      ;FOLD -- RSK Sammelstoerung -- ;%{SE}%MKUKATPVW %CVW_COM %VCOMMENT %P 2:-- RSK Sammelstoerung --, 3: VW_COMMENT
      ;ENDFOLD
      ;FOLD F329 = T7 + T9 + F325 ;%{SE}%MKUKATPVW %CVW_SPS %VBOASG %P 2:F329 = T7 + T9 + F325, 3: BOASG
         $FLAG[329] = $TIMER_FLAG[7] OR $TIMER_FLAG[9] OR $FLAG[325]
      ;ENDFOLD
      ;FOLD -- Hilfsflag Startfraesen -- ;%{SE}%MKUKATPVW %CVW_COM %VCOMMENT %P 2:-- Hilfsflag Startfraesen --, 3: VW_COMMENT
      ;ENDFOLD
      ;FOLD F152 = (F152 & F138 + F154 & F139) & F287 ;%{SE}%MKUKATPVW %CVW_SPS %VBOASG %P 2:F152 = (F152 & F138 + F154 & F139) & F287, 3: BOASG
         $FLAG[152] = ($FLAG[152] AND $FLAG[138] OR $FLAG[154] AND $FLAG[139]) AND $FLAG[287]
      ;ENDFOLD
      ;FOLD F154 = !F164 & F154 + F164 & F287 & F154 ;%{SE}%MKUKATPVW %CVW_SPS %VBOASG %P 2:F154 = !F164 & F154 + F164 & F287 & F154, 3: BOASG
         $FLAG[154] = NOT $FLAG[164] AND $FLAG[154] OR $FLAG[164] AND $FLAG[287] AND $FLAG[154]
      ;ENDFOLD
      ;FOLD F287 = F138 + F139 & F164 ;%{SE}%MKUKATPVW %CVW_SPS %VBOASG %P 2:F287 = F138 + F139 & F164, 3: BOASG
         $FLAG[287] = $FLAG[138] OR $FLAG[139] AND $FLAG[164]
      ;ENDFOLD
      ;FOLD -- Neues Fraesprogramm und Zaehler ruecksetzen -- ;%{SE}%MKUKATPVW %CVW_COM %VCOMMENT %P 2:-- Neues Fraesprogramm und Zaehler ruecksetzen --, 3: VW_COMMENT
      ;ENDFOLD
      ;FOLD bin3 ( F164 ) = 36 ;%{SE}%MKUKATPVW %CVW_SPS %VARIASG %P 2:bin3 ( F164 ) = 36, 3: ARIASG
         VW(#BINOUT,$FLAG[164],3,36)
      ;ENDFOLD
      ;FOLD i7 ( F152 ) = i45 ;%{SE}%MKUKATPVW %CVW_SPS %VARIASG %P 2:i7 ( F152 ) = i45, 3: ARIASG
         VW(#COUNTER,$FLAG[152],7,$COUNT_I[45])
      ;ENDFOLD
      ;FOLD -- Wiederholung beim Startfraesen -- ;%{SE}%MKUKATPVW %CVW_COM %VCOMMENT %P 2:-- Wiederholung beim Startfraesen --, 3: VW_COMMENT
      ;ENDFOLD
      ;FOLD Schritt 81 = E877 & !E878 & (F138 & !F152 + F139 & F164 & !F152) & !F325 & !F329 & A4039 ;%{SE}%MKUKATPVW %CVW_SPS %VST_CON %P 2:Schritt 81 = E877 & !E878 & (F138 & !F152 + F139 & F164 & !F152) & !F325 & !F329 & A4039, 3: ST_CON
         IF $IN[877] AND NOT $IN[878] AND ($FLAG[138] AND NOT $FLAG[152] OR $FLAG[139] AND $FLAG[164] AND NOT $FLAG[152]) AND NOT $FLAG[325] AND NOT $FLAG[329] AND $OUT[4039] THEN
            PREVSTEP = $APP_INT[5]
            $APP_INT[5] = 81
         ENDIF
      ;ENDFOLD
      ;FOLD -- Weiter wenn Fraesen fertig -- ;%{SE}%MKUKATPVW %CVW_COM %VCOMMENT %P 2:-- Weiter wenn Fraesen fertig --, 3: VW_COMMENT
      ;ENDFOLD
      ;FOLD Schritt 85 = E877 & !E878 & (F139 & F154 & (!F164 + F152) + F138 & F152 + F325 + F329) & A4039 ;%{SE}%MKUKATPVW %CVW_SPS %VST_CON %P 2:Schritt 85 = E877 & !E878 & (F139 & F154 & (!F164 + F152) + F138 & F152 + F325 + F329) & A4039, 3: ST_CON
         IF $IN[877] AND NOT $IN[878] AND ($FLAG[139] AND $FLAG[154] AND (NOT $FLAG[164] OR $FLAG[152]) OR $FLAG[138] AND $FLAG[152] OR $FLAG[325] OR $FLAG[329]) AND $OUT[4039] THEN
            PREVSTEP = $APP_INT[5]
            $APP_INT[5] = 85
         ENDIF
      ;ENDFOLD
   ;ENDFOLD
   ;FOLD SCHRITT 85 -- STAT EZ2/SP2/KE2-- ;%{P}%MKUKATPVW,%CSTEP,%VST_NR,%P 1:SCHRITT, 2:85, 3: STAT EZ2/SP2/KE2
      ;FOLD ;%{H}
         Case 85
      ;ENDFOLD
      ;FOLD F324 = AUS ;%{SE}%MKUKATPVW %CVW_SPS %VBOASG %P 2:F324 = AUS, 3: BOASG
         $FLAG[324] = FALSE
      ;ENDFOLD
      ;FOLD A877 = AUS ;%{SE}%MKUKATPVW %CVW_SPS %VBOASG %P 2:A877 = AUS, 3: BOASG
         $OUT[877] = FALSE
      ;ENDFOLD
      ;FOLD -- KF2 abschalten -- ;%{SE}%MKUKATPVW %CVW_COM %VCOMMENT %P 2:-- KF2 abschalten --, 3: VW_COMMENT
      ;ENDFOLD
      ;FOLD A994 = AUS ;%{SE}%MKUKATPVW %CVW_SPS %VBOASG %P 2:A994 = AUS, 3: BOASG
         $OUT[994] = FALSE
      ;ENDFOLD
      ;FOLD -- Ueberwachungszeit KF2 Versetzeinheit -- ;%{SE}%MKUKATPVW %CVW_COM %VCOMMENT %P 2:-- Ueberwachungszeit KF2 Versetzeinheit --, 3: VW_COMMENT
      ;ENDFOLD
      ;FOLD t8 ( EIN ) = -40[1/10Sek] ;%{SE}%MKUKATPVW %CVW_SPS %VTASG %P 2:t8 ( EIN ) = -40[1/10Sek], 3: TASG
         VW(#SET_TIME,TRUE,8,0,-40)
      ;ENDFOLD
      ;FOLD Schritt 86 = A4039 ;%{SE}%MKUKATPVW %CVW_SPS %VST_CON %P 2:Schritt 86 = A4039, 3: ST_CON
         IF $OUT[4039] THEN
            PREVSTEP = $APP_INT[5]
            $APP_INT[5] = 86
         ENDIF
      ;ENDFOLD
   ;ENDFOLD
   ;FOLD SCHRITT 86 -- STAT EZ2/SP2/KE2 -- ;%{P}%MKUKATPVW,%CSTEP,%VST_NR,%P 1:SCHRITT, 2:86, 3: STAT EZ2/SP2/KE2
      ;FOLD ;%{H}
         Case 86
      ;ENDFOLD
      ;FOLD F328 = AUS ;%{SE}%MKUKATPVW %CVW_SPS %VBOASG %P 2:F328 = AUS, 3: BOASG
         $FLAG[328] = FALSE
      ;ENDFOLD
      ;FOLD -- KF2 Versetzeinheit vor -- ;%{SE}%MKUKATPVW %CVW_COM %VCOMMENT %P 2:-- KF2 Versetzeinheit vor --, 3: VW_COMMENT
      ;ENDFOLD
      ;FOLD A995 = F565 ;%{SE}%MKUKATPVW %CVW_SPS %VBOASG %P 2:A995 = F565, 3: BOASG
         $OUT[995] = $FLAG[565]
      ;ENDFOLD
      ;FOLD -- RSK Fehlerausgabe KS2 Arbeitsst. -- ;%{SE}%MKUKATPVW %CVW_COM %VCOMMENT %P 2:-- RSK Fehlerausgabe KS2 Arbeitsst. --, 3: VW_COMMENT
      ;ENDFOLD
      ;FOLD F324 = (E996 + !E997 + !E998 + E999) & !F323 & !F328 + F324 ;%{SE}%MKUKATPVW %CVW_SPS %VBOASG %P 2:F324 = (E996 + !E997 + !E998 + E999) & !F323 & !F328 + F324, 3: BOASG
         $FLAG[324] = ($IN[996] OR NOT $IN[997] OR NOT $IN[998] OR $IN[999]) AND NOT $FLAG[323] AND NOT $FLAG[328] OR $FLAG[324]
      ;ENDFOLD
      ;FOLD -- RSK Sammelstoerung -- ;%{SE}%MKUKATPVW %CVW_COM %VCOMMENT %P 2:-- RSK Sammelstoerung --, 3: VW_COMMENT
      ;ENDFOLD
      ;FOLD F329 = F324 + F325 ;%{SE}%MKUKATPVW %CVW_SPS %VBOASG %P 2:F329 = F324 + F325, 3: BOASG
         $FLAG[329] = $FLAG[324] OR $FLAG[325]
      ;ENDFOLD
      ;FOLD -- Ueberwachungszeit KS2 schwenken -- ;%{SE}%MKUKATPVW %CVW_COM %VCOMMENT %P 2:-- Ueberwachungszeit KS2 schwenken --, 3: VW_COMMENT
      ;ENDFOLD
      ;FOLD t9 ( EIN ) = -100[1/10Sek] ;%{SE}%MKUKATPVW %CVW_SPS %VTASG %P 2:t9 ( EIN ) = -100[1/10Sek], 3: TASG
         VW(#SET_TIME,TRUE,9,0,-100)
      ;ENDFOLD
      ;FOLD Schritt 85 = F324 & (E26 + E27) & A4039 ;%{SE}%MKUKATPVW %CVW_SPS %VST_CON %P 2:Schritt 85 = F324 & (E26 + E27) & A4039, 3: ST_CON
         IF $FLAG[324] AND ($IN[26] OR $IN[27]) AND $OUT[4039] THEN
            PREVSTEP = $APP_INT[5]
            $APP_INT[5] = 85
         ENDIF
      ;ENDFOLD
      ;FOLD Schritt 87 = (!F324 & (E995 & F565 + !E995 & !F565) + T8 + F325) & A4039 ;%{SE}%MKUKATPVW %CVW_SPS %VST_CON %P 2:Schritt 87 = (!F324 & (E995 & F565 + !E995 & !F565) + T8 + F325) & A4039, 3: ST_CON
         IF (NOT $FLAG[324] AND ($IN[995] AND $FLAG[565] OR NOT $IN[995] AND NOT $FLAG[565]) OR $TIMER_FLAG[8] OR $FLAG[325]) AND $OUT[4039] THEN
            PREVSTEP = $APP_INT[5]
            $APP_INT[5] = 87
         ENDIF
      ;ENDFOLD
   ;ENDFOLD
   ;FOLD SCHRITT 87 -- STAT EZ2/SP2/KE2-- ;%{P}%MKUKATPVW,%CSTEP,%VST_NR,%P 1:SCHRITT, 2:87, 3: STAT EZ2/SP2/KE2
      ;FOLD ;%{H}
         Case 87
      ;ENDFOLD
      ;FOLD F323 = AUS ;%{SE}%MKUKATPVW %CVW_SPS %VBOASG %P 2:F323 = AUS, 3: BOASG
         $FLAG[323] = FALSE
      ;ENDFOLD
      ;FOLD F328 = AUS ;%{SE}%MKUKATPVW %CVW_SPS %VBOASG %P 2:F328 = AUS, 3: BOASG
         $FLAG[328] = FALSE
      ;ENDFOLD
      ;FOLD -- RSK Sammelstoerung -- ;%{SE}%MKUKATPVW %CVW_COM %VCOMMENT %P 2:-- RSK Sammelstoerung --, 3: VW_COMMENT
      ;ENDFOLD
      ;FOLD F329 = F325 ;%{SE}%MKUKATPVW %CVW_SPS %VBOASG %P 2:F329 = F325, 3: BOASG
         $FLAG[329] = $FLAG[325]
      ;ENDFOLD
      ;FOLD -- KF2 ein -- ;%{SE}%MKUKATPVW %CVW_COM %VCOMMENT %P 2:-- KF2 ein --, 3: VW_COMMENT
      ;ENDFOLD
      ;FOLD A994 = EIN ;%{SE}%MKUKATPVW %CVW_SPS %VBOASG %P 2:A994 = EIN, 3: BOASG
         $OUT[994] = TRUE
      ;ENDFOLD
      ;FOLD -- KS2 in Ruhestellung schwenken -- ;%{SE}%MKUKATPVW %CVW_COM %VCOMMENT %P 2:-- KS2 in Ruhestellung schwenken --, 3: VW_COMMENT
      ;ENDFOLD
      ;FOLD A1000 = (F746 + !F714) & E877 & (E995 & F565 + !E995 & !F565) ;%{SE}%MKUKATPVW %CVW_SPS %VBOASG %P 2:A1000 = (F746 + !F714) & E877 & (E995 & F565 + !E995 & !F565), 3: BOASG
         $OUT[1000] = ($FLAG[746] OR NOT $FLAG[714]) AND $IN[877] AND ($IN[995] AND $FLAG[565] OR NOT $IN[995] AND NOT $FLAG[565])
      ;ENDFOLD
      ;FOLD Schritt 88 = (F746 + !F714 + T9) & (A1000 + T9) & E877 & A4039 ;%{SE}%MKUKATPVW %CVW_SPS %VST_CON %P 2:Schritt 88 = (F746 + !F714 + T9) & (A1000 + T9) & E877 & A4039, 3: ST_CON
         IF ($FLAG[746] OR NOT $FLAG[714] OR $TIMER_FLAG[9]) AND ($OUT[1000] OR $TIMER_FLAG[9]) AND $IN[877] AND $OUT[4039] THEN
            PREVSTEP = $APP_INT[5]
            $APP_INT[5] = 88
         ENDIF
      ;ENDFOLD
   ;ENDFOLD
   ;FOLD SCHRITT 88 -- STAT EZ2/SP2/KE2 -- ;%{P}%MKUKATPVW,%CSTEP,%VST_NR,%P 1:SCHRITT, 2:88, 3: STAT EZ2/SP2/KE2
      ;FOLD ;%{H}
         Case 88
      ;ENDFOLD
      ;FOLD -- Hilfsflag SK Programmwechsel -- ;%{SE}%MKUKATPVW %CVW_COM %VCOMMENT %P 2:-- Hilfsflag SK Programmwechsel --, 3: VW_COMMENT
      ;ENDFOLD
      ;FOLD F334 = AUS ;%{SE}%MKUKATPVW %CVW_SPS %VBOASG %P 2:F334 = AUS, 3: BOASG
         $FLAG[334] = FALSE
      ;ENDFOLD
      ;FOLD -- RSK Fehlerausgabe KF Versetzeinheit -- ;%{SE}%MKUKATPVW %CVW_COM %VCOMMENT %P 2:-- RSK Fehlerausgabe KF Versetzeinheit --, 3: VW_COMMENT
      ;ENDFOLD
      ;FOLD F328 = !E995 & F565 & !F323 + F328 ;%{SE}%MKUKATPVW %CVW_SPS %VBOASG %P 2:F328 = !E995 & F565 & !F323 + F328, 3: BOASG
         $FLAG[328] = NOT $IN[995] AND $FLAG[565] AND NOT $FLAG[323] OR $FLAG[328]
      ;ENDFOLD
      ;FOLD -- RSK Fehlerausgabe KS2 Ruhestellung -- ;%{SE}%MKUKATPVW %CVW_COM %VCOMMENT %P 2:-- RSK Fehlerausgabe KS2 Ruhestellung --, 3: VW_COMMENT
      ;ENDFOLD
      ;FOLD F323 = (!E996 + E997 + E998 + !E999) & T9 & (E995 + !F565) + F323 ;%{SE}%MKUKATPVW %CVW_SPS %VBOASG %P 2:F323 = (!E996 + E997 + E998 + !E999) & T9 & (E995 + !F565) + F323, 3: BOASG
         $FLAG[323] = (NOT $IN[996] OR $IN[997] OR $IN[998] OR NOT $IN[999]) AND $TIMER_FLAG[9] AND ($IN[995] OR NOT $FLAG[565]) OR $FLAG[323]
      ;ENDFOLD
      ;FOLD -- RSK Fehlerausgabe EZ/SP min. Oeffnung -- ;%{SE}%MKUKATPVW %CVW_COM %VCOMMENT %P 2:-- RSK Fehlerausgabe EZ/SP min. Oeffnung --, 3: VW_COMMENT
      ;ENDFOLD
      ;FOLD F333 = !F746 ;%{SE}%MKUKATPVW %CVW_SPS %VBOASG %P 2:F333 = !F746, 3: BOASG
         $FLAG[333] = NOT $FLAG[746]
      ;ENDFOLD
      ;FOLD -- RSK Sammelstoerung -- ;%{SE}%MKUKATPVW %CVW_COM %VCOMMENT %P 2:-- RSK Sammelstoerung --, 3: VW_COMMENT
      ;ENDFOLD
      ;FOLD F329 = F323 + F325 + F328 + F333 ;%{SE}%MKUKATPVW %CVW_SPS %VBOASG %P 2:F329 = F323 + F325 + F328 + F333, 3: BOASG
         $FLAG[329] = $FLAG[323] OR $FLAG[325] OR $FLAG[328] OR $FLAG[333]
      ;ENDFOLD
      ;FOLD A994 = !F323 & !F328 ;%{SE}%MKUKATPVW %CVW_SPS %VBOASG %P 2:A994 = !F323 & !F328, 3: BOASG
         $OUT[994] = NOT $FLAG[323] AND NOT $FLAG[328]
      ;ENDFOLD
      ;FOLD A995 = F565 ;%{SE}%MKUKATPVW %CVW_SPS %VBOASG %P 2:A995 = F565, 3: BOASG
         $OUT[995] = $FLAG[565]
      ;ENDFOLD
      ;FOLD Schritt 86 = (F323 + F328) & (E26 + E27) & A4039 ;%{SE}%MKUKATPVW %CVW_SPS %VST_CON %P 2:Schritt 86 = (F323 + F328) & (E26 + E27) & A4039, 3: ST_CON
         IF ($FLAG[323] OR $FLAG[328]) AND ($IN[26] OR $IN[27]) AND $OUT[4039] THEN
            PREVSTEP = $APP_INT[5]
            $APP_INT[5] = 86
         ENDIF
      ;ENDFOLD
      ;FOLD Schritt 89 = !A1000 & E996 & !E997 & !E998 & E999 & A4039 ;%{SE}%MKUKATPVW %CVW_SPS %VST_CON %P 2:Schritt 89 = !A1000 & E996 & !E997 & !E998 & E999 & A4039, 3: ST_CON
         IF NOT $OUT[1000] AND $IN[996] AND NOT $IN[997] AND NOT $IN[998] AND $IN[999] AND $OUT[4039] THEN
            PREVSTEP = $APP_INT[5]
            $APP_INT[5] = 89
         ENDIF
      ;ENDFOLD
   ;ENDFOLD
   ;FOLD SCHRITT 89 -- STAT EZ2/SP2/KE2 -- ;%{P}%MKUKATPVW,%CSTEP,%VST_NR,%P 1:SCHRITT, 2:89, 3: STAT EZ2/SP2/KE2
      ;FOLD ;%{H}
         Case 89
      ;ENDFOLD
      ;FOLD F323 = AUS ;%{SE}%MKUKATPVW %CVW_SPS %VBOASG %P 2:F323 = AUS, 3: BOASG
         $FLAG[323] = FALSE
      ;ENDFOLD
      ;FOLD F328 = AUS ;%{SE}%MKUKATPVW %CVW_SPS %VBOASG %P 2:F328 = AUS, 3: BOASG
         $FLAG[328] = FALSE
      ;ENDFOLD
      ;FOLD -- RSK Sammelstoerung -- ;%{SE}%MKUKATPVW %CVW_COM %VCOMMENT %P 2:-- RSK Sammelstoerung --, 3: VW_COMMENT
      ;ENDFOLD
      ;FOLD F329 = F325 ;%{SE}%MKUKATPVW %CVW_SPS %VBOASG %P 2:F329 = F325, 3: BOASG
         $FLAG[329] = $FLAG[325]
      ;ENDFOLD
      ;FOLD t9 ( EIN ) = STOP ;%{SE}%MKUKATPVW %CVW_SPS %VTSTOP %P 2:t9 ( EIN ) = STOP, 3: TSTOP
         VW(#SET_TIME,TRUE,9,1,0)
      ;ENDFOLD
      ;FOLD -- KF2 Versetzeinheit rueck -- ;%{SE}%MKUKATPVW %CVW_COM %VCOMMENT %P 2:-- KF2 Versetzeinheit rueck --, 3: VW_COMMENT
      ;ENDFOLD
      ;FOLD A995 = AUS ;%{SE}%MKUKATPVW %CVW_SPS %VBOASG %P 2:A995 = AUS, 3: BOASG
         $OUT[995] = FALSE
      ;ENDFOLD
      ;FOLD -- KF2 aus -- ;%{SE}%MKUKATPVW %CVW_COM %VCOMMENT %P 2:-- KF2 aus --, 3: VW_COMMENT
      ;ENDFOLD
      ;FOLD A994 = AUS ;%{SE}%MKUKATPVW %CVW_SPS %VBOASG %P 2:A994 = AUS, 3: BOASG
         $OUT[994] = FALSE
      ;ENDFOLD
      ;FOLD -- KF1 Ausblasen -- ;%{SE}%MKUKATPVW %CVW_COM %VCOMMENT %P 2:-- KF1 Ausblasen --, 3: VW_COMMENT
      ;ENDFOLD
      ;FOLD A996 = (F330 + F331 + F332) & F738 ;%{SE}%MKUKATPVW %CVW_SPS %VBOASG %P 2:A996 = (F330 + F331 + F332) & F738, 3: BOASG
         $OUT[996] = ($FLAG[330] OR $FLAG[331] OR $FLAG[332]) AND $FLAG[738]
      ;ENDFOLD
      ;FOLD bin3 ( F285 ) = 5 ;%{SE}%MKUKATPVW %CVW_SPS %VARIASG %P 2:bin3 ( F285 ) = 5, 3: ARIASG
         VW(#BINOUT,$FLAG[285],3,5)
      ;ENDFOLD
      ;FOLD bin6 ( !F285 ) = 1 ;%{SE}%MKUKATPVW %CVW_SPS %VARIASG %P 2:bin6 ( !F285 ) = 1, 3: ARIASG
         VW(#BINOUT,NOT $FLAG[285],6,1)
      ;ENDFOLD
      ;FOLD -- Wartezeit Programmwechsel SK -- ;%{SE}%MKUKATPVW %CVW_COM %VCOMMENT %P 2:-- Wartezeit Programmwechsel SK --, 3: VW_COMMENT
      ;ENDFOLD
      ;FOLD T8 ( !F334 ) = -2[1/10Sek] ;%{SE}%MKUKATPVW %CVW_SPS %VTASG %P 2:T8 ( !F334 ) = -2[1/10Sek], 3: TASG
         VW(#SET_TIME,NOT $FLAG[334],8,0,-2)
      ;ENDFOLD
      ;FOLD -- Hilfsflag SK Programmwechsel -- ;%{SE}%MKUKATPVW %CVW_COM %VCOMMENT %P 2:-- Hilfsflag SK Programmwechsel --, 3: VW_COMMENT
      ;ENDFOLD
      ;FOLD F334 = EIN ;%{SE}%MKUKATPVW %CVW_SPS %VBOASG %P 2:F334 = EIN, 3: BOASG
         $FLAG[334] = TRUE
      ;ENDFOLD
      ;FOLD -- Ueberwachungszeit EZ2/SP2/KE2 Messen -- ;%{SE}%MKUKATPVW %CVW_COM %VCOMMENT %P 2:-- Ueberwachungszeit EZ2/SP2/KE2 Messen --, 3: VW_COMMENT
      ;ENDFOLD
      ;FOLD t9 ( EIN ) = -150[1/10Sek] ;%{SE}%MKUKATPVW %CVW_SPS %VTASG %P 2:t9 ( EIN ) = -150[1/10Sek], 3: TASG
         VW(#SET_TIME,TRUE,9,0,-150)
      ;ENDFOLD
      ;FOLD Schritt 74 = (F325 + F329) & (E26 + E27) & A4039 ;%{SE}%MKUKATPVW %CVW_SPS %VST_CON %P 2:Schritt 74 = (F325 + F329) & (E26 + E27) & A4039, 3: ST_CON
         IF ($FLAG[325] OR $FLAG[329]) AND ($IN[26] OR $IN[27]) AND $OUT[4039] THEN
            PREVSTEP = $APP_INT[5]
            $APP_INT[5] = 74
         ENDIF
      ;ENDFOLD
      ;FOLD Schritt 90 = T8 & !F325 & !F329 & A4039 ;%{SE}%MKUKATPVW %CVW_SPS %VST_CON %P 2:Schritt 90 = T8 & !F325 & !F329 & A4039, 3: ST_CON
         IF $TIMER_FLAG[8] AND NOT $FLAG[325] AND NOT $FLAG[329] AND $OUT[4039] THEN
            PREVSTEP = $APP_INT[5]
            $APP_INT[5] = 90
         ENDIF
      ;ENDFOLD
   ;ENDFOLD
   ;FOLD SCHRITT 90 -- STAT EZ2/SP2/KE2 -- ;%{P}%MKUKATPVW,%CSTEP,%VST_NR,%P 1:SCHRITT, 2:90, 3: STAT EZ2/SP2/KE2
      ;FOLD ;%{H}
         Case 90
      ;ENDFOLD
      ;FOLD -- Hilfsflag SK Programmwechsel -- ;%{SE}%MKUKATPVW %CVW_COM %VCOMMENT %P 2:-- Hilfsflag SK Programmwechsel --, 3: VW_COMMENT
      ;ENDFOLD
      ;FOLD F334 = AUS ;%{SE}%MKUKATPVW %CVW_SPS %VBOASG %P 2:F334 = AUS, 3: BOASG
         $FLAG[334] = FALSE
      ;ENDFOLD
      ;FOLD -- Quitt. Fraesen SK2/SK1 -- ;%{SE}%MKUKATPVW %CVW_COM %VCOMMENT %P 2:-- Quitt. Fraesen SK2/SK1 --, 3: VW_COMMENT
      ;ENDFOLD
      ;FOLD A946 = !F285 & !F329 & !F322 ;%{SE}%MKUKATPVW %CVW_SPS %VBOASG %P 2:A946 = !F285 & !F329 & !F322, 3: BOASG
         $OUT[946] = NOT $FLAG[285] AND NOT $FLAG[329] AND NOT $FLAG[322]
      ;ENDFOLD
      ;FOLD A786 = F285 & !F329 & !F322 ;%{SE}%MKUKATPVW %CVW_SPS %VBOASG %P 2:A786 = F285 & !F329 & !F322, 3: BOASG
         $OUT[786] = $FLAG[285] AND NOT $FLAG[329] AND NOT $FLAG[322]
      ;ENDFOLD
      ;FOLD -- RSK Sammelstoerung -- ;%{SE}%MKUKATPVW %CVW_COM %VCOMMENT %P 2:-- RSK Sammelstoerung --, 3: VW_COMMENT
      ;ENDFOLD
      ;FOLD F329 = T9 ;%{SE}%MKUKATPVW %CVW_SPS %VBOASG %P 2:F329 = T9, 3: BOASG
         $FLAG[329] = $TIMER_FLAG[9]
      ;ENDFOLD
      ;FOLD -- Messen nach Fraesen -- ;%{SE}%MKUKATPVW %CVW_COM %VCOMMENT %P 2:-- Messen nach Fraesen --, 3: VW_COMMENT
      ;ENDFOLD
      ;FOLD A919 = !F138 & F139 ;%{SE}%MKUKATPVW %CVW_SPS %VBOASG %P 2:A919 = !F138 & F139, 3: BOASG
         $OUT[919] = NOT $FLAG[138] AND $FLAG[139]
      ;ENDFOLD
      ;FOLD A918 = F138 & !F139 ;%{SE}%MKUKATPVW %CVW_SPS %VBOASG %P 2:A918 = F138 & !F139, 3: BOASG
         $OUT[918] = $FLAG[138] AND NOT $FLAG[139]
      ;ENDFOLD
      ;FOLD A917 = (F138 + F139) & !F329 ;%{SE}%MKUKATPVW %CVW_SPS %VBOASG %P 2:A917 = (F138 + F139) & !F329, 3: BOASG
         $OUT[917] = ($FLAG[138] OR $FLAG[139]) AND NOT $FLAG[329]
      ;ENDFOLD
      ;FOLD Schritt 91 = (!E946 & E947 & !E948 + F285 & !E786 & E787 & !E788) & A4039 ;%{SE}%MKUKATPVW %CVW_SPS %VST_CON %P 2:Schritt 91 = (!E946 & E947 & !E948 + F285 & !E786 & E787 & !E788) & A4039, 3: ST_CON
         IF (NOT $IN[946] AND $IN[947] AND NOT $IN[948] OR $FLAG[285] AND NOT $IN[786] AND $IN[787] AND NOT $IN[788]) AND $OUT[4039] THEN
            PREVSTEP = $APP_INT[5]
            $APP_INT[5] = 91
         ENDIF
      ;ENDFOLD
   ;ENDFOLD
   ;FOLD SCHRITT 91 -- STAT EZ2/SP2/KE2 -- ;%{P}%MKUKATPVW,%CSTEP,%VST_NR,%P 1:SCHRITT, 2:91, 3: STAT EZ2/SP2/KE2
      ;FOLD ;%{H}
         Case 91
      ;ENDFOLD
      ;FOLD -- Hilfsflag SK Programmwechsel -- ;%{SE}%MKUKATPVW %CVW_COM %VCOMMENT %P 2:-- Hilfsflag SK Programmwechsel --, 3: VW_COMMENT
      ;ENDFOLD
      ;FOLD F334 = AUS ;%{SE}%MKUKATPVW %CVW_SPS %VBOASG %P 2:F334 = AUS, 3: BOASG
         $FLAG[334] = FALSE
      ;ENDFOLD
      ;FOLD -- RSK Sammelstoerung -- ;%{SE}%MKUKATPVW %CVW_COM %VCOMMENT %P 2:-- RSK Sammelstoerung --, 3: VW_COMMENT
      ;ENDFOLD
      ;FOLD F329 = T9 ;%{SE}%MKUKATPVW %CVW_SPS %VBOASG %P 2:F329 = T9, 3: BOASG
         $FLAG[329] = $TIMER_FLAG[9]
      ;ENDFOLD
      ;FOLD Schritt 92 = E877 & (E917 & !E936 + T9) & A4039 ;%{SE}%MKUKATPVW %CVW_SPS %VST_CON %P 2:Schritt 92 = E877 & (E917 & !E936 + T9) & A4039, 3: ST_CON
         IF $IN[877] AND ($IN[917] AND NOT $IN[936] OR $TIMER_FLAG[9]) AND $OUT[4039] THEN
            PREVSTEP = $APP_INT[5]
            $APP_INT[5] = 92
         ENDIF
      ;ENDFOLD
   ;ENDFOLD
   ;FOLD SCHRITT 92 -- STAT EZ2/SP2/KE2-- ;%{P}%MKUKATPVW,%CSTEP,%VST_NR,%P 1:SCHRITT, 2:92, 3: STAT EZ2/SP2/KE2
      ;FOLD ;%{H}
         Case 92
      ;ENDFOLD
      ;FOLD -- RSK Fehlerausgabe Kappenverschleiss -- ;%{SE}%MKUKATPVW %CVW_COM %VCOMMENT %P 2:-- RSK Fehlerausgabe Kappenverschleiss --, 3: VW_COMMENT
      ;ENDFOLD
      ;FOLD F160 = E937 ;%{SE}%MKUKATPVW %CVW_SPS %VBOASG %P 2:F160 = E937, 3: BOASG
         $FLAG[160] = $IN[937]
      ;ENDFOLD
      ;FOLD -- RSK Fehlerausgabe Messen -- ;%{SE}%MKUKATPVW %CVW_COM %VCOMMENT %P 2:-- RSK Fehlerausgabe Messen --, 3: VW_COMMENT
      ;ENDFOLD
      ;FOLD F326 = E936 + E937 + E938 + F326 ;%{SE}%MKUKATPVW %CVW_SPS %VBOASG %P 2:F326 = E936 + E937 + E938 + F326, 3: BOASG
         $FLAG[326] = $IN[936] OR $IN[937] OR $IN[938] OR $FLAG[326]
      ;ENDFOLD
      ;FOLD -- RSK Sammelstoerung -- ;%{SE}%MKUKATPVW %CVW_COM %VCOMMENT %P 2:-- RSK Sammelstoerung --, 3: VW_COMMENT
      ;ENDFOLD
      ;FOLD F329 = F326 ;%{SE}%MKUKATPVW %CVW_SPS %VBOASG %P 2:F329 = F326, 3: BOASG
         $FLAG[329] = $FLAG[326]
      ;ENDFOLD
      ;FOLD A918 = AUS ;%{SE}%MKUKATPVW %CVW_SPS %VBOASG %P 2:A918 = AUS, 3: BOASG
         $OUT[918] = FALSE
      ;ENDFOLD
      ;FOLD A919 = AUS ;%{SE}%MKUKATPVW %CVW_SPS %VBOASG %P 2:A919 = AUS, 3: BOASG
         $OUT[919] = FALSE
      ;ENDFOLD
      ;FOLD -- Hilfsflag Startfrasen EZ2/SP2/KE2 an SK1 -- ;%{SE}%MKUKATPVW %CVW_COM %VCOMMENT %P 2:-- Hilfsflag Startfrasen EZ2/SP2/KE2 an SK1 --, 3: VW_COMMENT
      ;ENDFOLD
      ;FOLD F307 = F285 & F138 ;%{SE}%MKUKATPVW %CVW_SPS %VBOASG %P 2:F307 = F285 & F138, 3: BOASG
         $FLAG[307] = $FLAG[285] AND $FLAG[138]
      ;ENDFOLD
      ;FOLD -- Hilfsflag Normalfrasen EZ2/SP2/KE2 an SK1 -- ;%{SE}%MKUKATPVW %CVW_COM %VCOMMENT %P 2:-- Hilfsflag Normalfrasen EZ2/SP2/KE2 an SK1 --, 3: VW_COMMENT
      ;ENDFOLD
      ;FOLD F308 = F285 & F139 ;%{SE}%MKUKATPVW %CVW_SPS %VBOASG %P 2:F308 = F285 & F139, 3: BOASG
         $FLAG[308] = $FLAG[285] AND $FLAG[139]
      ;ENDFOLD
      ;FOLD -- Ueberwachungszeit EZ2/SP2/KE2 Setzhub 2 -- ;%{SE}%MKUKATPVW %CVW_COM %VCOMMENT %P 2:-- Ueberwachungszeit EZ2/SP2/KE2 Setzhub 2 --, 3: VW_COMMENT
      ;ENDFOLD
      ;FOLD t9 ( EIN ) = -80[1/10Sek] ;%{SE}%MKUKATPVW %CVW_SPS %VTASG %P 2:t9 ( EIN ) = -80[1/10Sek], 3: TASG
         VW(#SET_TIME,TRUE,9,0,-80)
      ;ENDFOLD
      ;FOLD -- Druckvorgabe SK2/SK1/EZ2/SP2/KE2 -- ;%{SE}%MKUKATPVW %CVW_COM %VCOMMENT %P 2:-- Druckvorgabe SK2/SK1/EZ2/SP2/KE2 --, 3: VW_COMMENT
      ;ENDFOLD
      ;FOLD bin3 (F307) = 45 ;%{SE}%MKUKATPVW %CVW_SPS %VARIASG %P 2:bin3 (F307) = 45, 3: ARIASG
         VW(#BINOUT,$FLAG[307],3,45)
      ;ENDFOLD
      ;FOLD bin3 (F308) = 55 ;%{SE}%MKUKATPVW %CVW_SPS %VARIASG %P 2:bin3 (F308) = 55, 3: ARIASG
         VW(#BINOUT,$FLAG[308],3,55)
      ;ENDFOLD
      ;FOLD F168 = F138 & !F831 ;%{SE}%MKUKATPVW %CVW_SPS %VBOASG %P 2:F168 = F138 & !F831, 3: BOASG
         $FLAG[168] = $FLAG[138] AND NOT $FLAG[831]
      ;ENDFOLD
      ;FOLD bin4 (F168) = 41 ;%{SE}%MKUKATPVW %CVW_SPS %VARIASG %P 2:bin4 (F168) = 41, 3: ARIASG
         VW(#BINOUT,$FLAG[168],4,41)
      ;ENDFOLD
      ;FOLD F168 = F139 & !F831 ;%{SE}%MKUKATPVW %CVW_SPS %VBOASG %P 2:F168 = F139 & !F831, 3: BOASG
         $FLAG[168] = $FLAG[139] AND NOT $FLAG[831]
      ;ENDFOLD
      ;FOLD bin4 (F168) = 51 ;%{SE}%MKUKATPVW %CVW_SPS %VARIASG %P 2:bin4 (F168) = 51, 3: ARIASG
         VW(#BINOUT,$FLAG[168],4,51)
      ;ENDFOLD
      ;FOLD F168 = AUS ;%{SE}%MKUKATPVW %CVW_SPS %VBOASG %P 2:F168 = AUS, 3: BOASG
         $FLAG[168] = FALSE
      ;ENDFOLD
      ;FOLD bin6 (F138) = 41 ;%{SE}%MKUKATPVW %CVW_SPS %VARIASG %P 2:bin6 (F138) = 41, 3: ARIASG
         VW(#BINOUT,$FLAG[138],6,41)
      ;ENDFOLD
      ;FOLD bin6 (F139) = 51 ;%{SE}%MKUKATPVW %CVW_SPS %VARIASG %P 2:bin6 (F139) = 51, 3: ARIASG
         VW(#BINOUT,$FLAG[139],6,51)
      ;ENDFOLD
      ;FOLD -- Wartezeit Programmwechsel SK -- ;%{SE}%MKUKATPVW %CVW_COM %VCOMMENT %P 2:-- Wartezeit Programmwechsel SK --, 3: VW_COMMENT
      ;ENDFOLD
      ;FOLD T8 ( !F334 ) = -2[1/10Sek] ;%{SE}%MKUKATPVW %CVW_SPS %VTASG %P 2:T8 ( !F334 ) = -2[1/10Sek], 3: TASG
         VW(#SET_TIME,NOT $FLAG[334],8,0,-2)
      ;ENDFOLD
      ;FOLD -- Hilfsflag SK Programmwechsel -- ;%{SE}%MKUKATPVW %CVW_COM %VCOMMENT %P 2:-- Hilfsflag SK Programmwechsel --, 3: VW_COMMENT
      ;ENDFOLD
      ;FOLD F334 = EIN ;%{SE}%MKUKATPVW %CVW_SPS %VBOASG %P 2:F334 = EIN, 3: BOASG
         $FLAG[334] = TRUE
      ;ENDFOLD
      ;FOLD Schritt 93 = T8 & !F335 & A4039 ;%{SE}%MKUKATPVW %CVW_SPS %VST_CON %P 2:Schritt 93 = T8 & !F335 & A4039, 3: ST_CON
         IF $TIMER_FLAG[8] AND NOT $FLAG[335] AND $OUT[4039] THEN
            PREVSTEP = $APP_INT[5]
            $APP_INT[5] = 93
         ENDIF
      ;ENDFOLD
      ;FOLD Schritt 93 = T8 & F335 & !F138 & !F307 & A4039 ;%{SE}%MKUKATPVW %CVW_SPS %VST_CON %P 2:Schritt 93 = T8 & F335 & !F138 & !F307 & A4039, 3: ST_CON
         IF $TIMER_FLAG[8] AND $FLAG[335] AND NOT $FLAG[138] AND NOT $FLAG[307] AND $OUT[4039] THEN
            PREVSTEP = $APP_INT[5]
            $APP_INT[5] = 93
         ENDIF
      ;ENDFOLD
      ;FOLD Schritt 222 = T8 & F335 & (F307 + F138) & A4039 ;%{SE}%MKUKATPVW %CVW_SPS %VST_CON %P 2:Schritt 222 = T8 & F335 & (F307 + F138) & A4039, 3: ST_CON
         IF $TIMER_FLAG[8] AND $FLAG[335] AND ($FLAG[307] OR $FLAG[138]) AND $OUT[4039] THEN
            PREVSTEP = $APP_INT[5]
            $APP_INT[5] = 222
         ENDIF
      ;ENDFOLD
   ;ENDFOLD
   ;FOLD SCHRITT 93 -- STAT EZ2/SP2/KE2 -- ;%{P}%MKUKATPVW,%CSTEP,%VST_NR,%P 1:SCHRITT, 2:93, 3: STAT EZ2/SP2/KE2
      ;FOLD ;%{H}
         Case 93
      ;ENDFOLD
      ;FOLD -- Hilfsflag SK Programmwechsel -- ;%{SE}%MKUKATPVW %CVW_COM %VCOMMENT %P 2:-- Hilfsflag SK Programmwechsel --, 3: VW_COMMENT
      ;ENDFOLD
      ;FOLD F334 = AUS ;%{SE}%MKUKATPVW %CVW_SPS %VBOASG %P 2:F334 = AUS, 3: BOASG
         $FLAG[334] = FALSE
      ;ENDFOLD
      ;FOLD A917 = AUS ;%{SE}%MKUKATPVW %CVW_SPS %VBOASG %P 2:A917 = AUS, 3: BOASG
         $OUT[917] = FALSE
      ;ENDFOLD
      ;FOLD -- EZ2/SP2/KE2 schliessen -- ;%{SE}%MKUKATPVW %CVW_COM %VCOMMENT %P 2:-- EZ2/SP2/KE2 schliessen --, 3: VW_COMMENT
      ;ENDFOLD
      ;FOLD A877 = AUS ;%{SE}%MKUKATPVW %CVW_SPS %VBOASG %P 2:A877 = AUS, 3: BOASG
         $OUT[877] = FALSE
      ;ENDFOLD
      ;FOLD A878 = !F329 & !F160 ;%{SE}%MKUKATPVW %CVW_SPS %VBOASG %P 2:A878 = !F329 & !F160, 3: BOASG
         $OUT[878] = NOT $FLAG[329] AND NOT $FLAG[160]
      ;ENDFOLD
      ;FOLD -- Ueberwachungszeit Kurzschlussschweissung SK2/SK1 -- ;%{SE}%MKUKATPVW %CVW_COM %VCOMMENT %P 2:-- Ueberwachungszeit Kurzschlussschweissung SK2/SK1 --, 3: VW_COMMENT
      ;ENDFOLD
      ;FOLD t9 ( EIN ) = -80[1/10Sek] ;%{SE}%MKUKATPVW %CVW_SPS %VTASG %P 2:t9 ( EIN ) = -80[1/10Sek], 3: TASG
         VW(#SET_TIME,TRUE,9,0,-80)
      ;ENDFOLD
      ;FOLD Schritt 94 = F285 & A514 & !E877 & E878 + E877 & !E878 & (F329 + F326 + F160) & A4039 ;%{SE}%MKUKATPVW %CVW_SPS %VST_CON %P 2:Schritt 94 = F285 & A514 & !E877 & E878 + E877 & !E878 & (F329 + F326 + F160) & A4039, 3: ST_CON
         IF $FLAG[285] AND $OUT[514] AND NOT $IN[877] AND $IN[878] OR $IN[877] AND NOT $IN[878] AND ($FLAG[329] OR $FLAG[326] OR $FLAG[160]) AND $OUT[4039] THEN
            PREVSTEP = $APP_INT[5]
            $APP_INT[5] = 94
         ENDIF
      ;ENDFOLD
      ;FOLD Schritt 94 = !F285 & !A514 & !E877 & E878 + E877 & !E878 & (F329 + F326 + F160) & A4039 ;%{SE}%MKUKATPVW %CVW_SPS %VST_CON %P 2:Schritt 94 = !F285 & !A514 & !E877 & E878 + E877 & !E878 & (F329 + F326 + F160) & A4039, 3: ST_CON
         IF NOT $FLAG[285] AND NOT $OUT[514] AND NOT $IN[877] AND $IN[878] OR $IN[877] AND NOT $IN[878] AND ($FLAG[329] OR $FLAG[326] OR $FLAG[160]) AND $OUT[4039] THEN
            PREVSTEP = $APP_INT[5]
            $APP_INT[5] = 94
         ENDIF
      ;ENDFOLD
   ;ENDFOLD
   ;FOLD SCHRITT 94 -- STAT EZ2/SP2/KE2-- ;%{P}%MKUKATPVW,%CSTEP,%VST_NR,%P 1:SCHRITT, 2:94, 3: STAT EZ2/SP2/KE2
      ;FOLD ;%{H}
         Case 94
      ;ENDFOLD
      ;FOLD -- Hilfsflag SK Programmwechsel -- ;%{SE}%MKUKATPVW %CVW_COM %VCOMMENT %P 2:-- Hilfsflag SK Programmwechsel --, 3: VW_COMMENT
      ;ENDFOLD
      ;FOLD F334 = AUS ;%{SE}%MKUKATPVW %CVW_SPS %VBOASG %P 2:F334 = AUS, 3: BOASG
         $FLAG[334] = FALSE
      ;ENDFOLD
      ;FOLD t9 ( EIN ) = STOP ;%{SE}%MKUKATPVW %CVW_SPS %VTSTOP %P 2:t9 ( EIN ) = STOP, 3: TSTOP
         VW(#SET_TIME,TRUE,9,1,0)
      ;ENDFOLD
      ;FOLD -- RSK Fehlerausgabe EZ2/SP2/KE2 Kraftaufbau -- ;%{SE}%MKUKATPVW %CVW_COM %VCOMMENT %P 2:-- RSK Fehlerausgabe EZ2/SP2/KE2 Kraftaufbau --, 3: VW_COMMENT
      ;ENDFOLD
      ;FOLD F325 = T9 + F325 ;%{SE}%MKUKATPVW %CVW_SPS %VBOASG %P 2:F325 = T9 + F325, 3: BOASG
         $FLAG[325] = $TIMER_FLAG[9] OR $FLAG[325]
      ;ENDFOLD
      ;FOLD -- RSK Fehlerausgabe K -- ;%{SE}%MKUKATPVW %CVW_COM %VCOMMENT %P 2:-- RSK Fehlerausgabe K --, 3: VW_COMMENT
      ;ENDFOLD
      ;FOLD F327 = (A785 & !F830 + A718 & F830) & (E805 + !E802) + F327 ;%{SE}%MKUKATPVW %CVW_SPS %VBOASG %P 2:F327 = (A785 & !F830 + A718 & F830) & (E805 + !E802) + F327, 3: BOASG
         $FLAG[327] = ($OUT[785] AND NOT $FLAG[830] OR $OUT[718] AND $FLAG[830]) AND ($IN[805] OR NOT $IN[802]) OR $FLAG[327]
      ;ENDFOLD
      ;FOLD F327 = (A945 & !F831 + A878 & F831) & (E965 + !E962) + F327 ;%{SE}%MKUKATPVW %CVW_SPS %VBOASG %P 2:F327 = (A945 & !F831 + A878 & F831) & (E965 + !E962) + F327, 3: BOASG
         $FLAG[327] = ($OUT[945] AND NOT $FLAG[831] OR $OUT[878] AND $FLAG[831]) AND ($IN[965] OR NOT $IN[962]) OR $FLAG[327]
      ;ENDFOLD
      ;FOLD -- RSK Sammelstoerung -- ;%{SE}%MKUKATPVW %CVW_COM %VCOMMENT %P 2:-- RSK Sammelstoerung --, 3: VW_COMMENT
      ;ENDFOLD
      ;FOLD F329 = F325 + F326 + F327 ;%{SE}%MKUKATPVW %CVW_SPS %VBOASG %P 2:F329 = F325 + F326 + F327, 3: BOASG
         $FLAG[329] = $FLAG[325] OR $FLAG[326] OR $FLAG[327]
      ;ENDFOLD
      ;FOLD -- Kurzschlussschweissung SK2/SK1 -- ;%{SE}%MKUKATPVW %CVW_COM %VCOMMENT %P 2:-- Kurzschlussschweissung SK2/SK1 --, 3: VW_COMMENT
      ;ENDFOLD
      ;FOLD A945 = !F285 & !F325 & !F329 & !F160 ;%{SE}%MKUKATPVW %CVW_SPS %VBOASG %P 2:A945 = !F285 & !F325 & !F329 & !F160, 3: BOASG
         $OUT[945] = NOT $FLAG[285] AND NOT $FLAG[325] AND NOT $FLAG[329] AND NOT $FLAG[160]
      ;ENDFOLD
      ;FOLD A785 = F285 & !F325 & !F329 & !F160 + !F285 & A785 ;%{SE}%MKUKATPVW %CVW_SPS %VBOASG %P 2:A785 = F285 & !F325 & !F329 & !F160 + !F285 & A785, 3: BOASG
         $OUT[785] = $FLAG[285] AND NOT $FLAG[325] AND NOT $FLAG[329] AND NOT $FLAG[160] OR NOT $FLAG[285] AND $OUT[785]
      ;ENDFOLD
      ;FOLD -- Flagbildung Wiederholfraesen -- ;%{SE}%MKUKATPVW %CVW_COM %VCOMMENT %P 2:-- Flagbildung Wiederholfraesen --, 3: VW_COMMENT
      ;ENDFOLD
      ;FOLD F749 = (F322 + F323 + F325 + F326 + F327 + F329) & !F748 ;%{SE}%MKUKATPVW %CVW_SPS %VBOASG %P 2:F749 = (F322 + F323 + F325 + F326 + F327 + F329) & !F748, 3: BOASG
         $FLAG[749] = ($FLAG[322] OR $FLAG[323] OR $FLAG[325] OR $FLAG[326] OR $FLAG[327] OR $FLAG[329]) AND NOT $FLAG[748]
      ;ENDFOLD
      ;FOLD Schritt 74 = E877 & !E878 & (F322 + F323 + F325 + F326 + F327 + F329) & (E26 + E27) & A4039 ;%{SE}%MKUKATPVW %CVW_SPS %VST_CON %P 2:Schritt 74 = E877 & !E878 & (F322 + F323 + F325 + F326 + F327 + F329) & (E26 + E27) & A4039, 3: ST_CON
         IF $IN[877] AND NOT $IN[878] AND ($FLAG[322] OR $FLAG[323] OR $FLAG[325] OR $FLAG[326] OR $FLAG[327] OR $FLAG[329]) AND ($IN[26] OR $IN[27]) AND $OUT[4039] THEN
            PREVSTEP = $APP_INT[5]
            $APP_INT[5] = 74
         ENDIF
      ;ENDFOLD
      ;FOLD Schritt 95 = (!F285 & E945 & E964 + F285 & E785 & E804 + F326 + F327 + F160) & A4039 ;%{SE}%MKUKATPVW %CVW_SPS %VST_CON %P 2:Schritt 95 = (!F285 & E945 & E964 + F285 & E785 & E804 + F326 + F327 + F160) & A4039, 3: ST_CON
         IF (NOT $FLAG[285] AND $IN[945] AND $IN[964] OR $FLAG[285] AND $IN[785] AND $IN[804] OR $FLAG[326] OR $FLAG[327] OR $FLAG[160]) AND $OUT[4039] THEN
            PREVSTEP = $APP_INT[5]
            $APP_INT[5] = 95
         ENDIF
      ;ENDFOLD
      ;FOLD Schritt 95 = (!F285 & E945 & E15 + F285 & E785 & E15 + F326 + F327 + F160) & A4039 ;%{SE}%MKUKATPVW %CVW_SPS %VST_CON %P 2:Schritt 95 = (!F285 & E945 & E15 + F285 & E785 & E15 + F326 + F327 + F160) & A4039, 3: ST_CON
         IF (NOT $FLAG[285] AND $IN[945] AND $IN[15] OR $FLAG[285] AND $IN[785] AND $IN[15] OR $FLAG[326] OR $FLAG[327] OR $FLAG[160]) AND $OUT[4039] THEN
            PREVSTEP = $APP_INT[5]
            $APP_INT[5] = 95
         ENDIF
      ;ENDFOLD
   ;ENDFOLD
   ;FOLD SCHRITT 95 -- STAT EZ2/SP2/KE2 -- ;%{P}%MKUKATPVW,%CSTEP,%VST_NR,%P 1:SCHRITT, 2:95, 3: STAT EZ2/SP2/KE2
      ;FOLD ;%{H}
         Case 95
      ;ENDFOLD
      ;FOLD A945 = AUS ;%{SE}%MKUKATPVW %CVW_SPS %VBOASG %P 2:A945 = AUS, 3: BOASG
         $OUT[945] = FALSE
      ;ENDFOLD
      ;FOLD A785 = F285 & !E785 + !F285 & A785 ;%{SE}%MKUKATPVW %CVW_SPS %VBOASG %P 2:A785 = F285 & !E785 + !F285 & A785, 3: BOASG
         $OUT[785] = $FLAG[285] AND NOT $IN[785] OR NOT $FLAG[285] AND $OUT[785]
      ;ENDFOLD
      ;FOLD F138 = !F327 & F138 ;%{SE}%MKUKATPVW %CVW_SPS %VBOASG %P 2:F138 = !F327 & F138, 3: BOASG
         $FLAG[138] = NOT $FLAG[327] AND $FLAG[138]
      ;ENDFOLD
      ;FOLD F139 = F327 + F139 ;%{SE}%MKUKATPVW %CVW_SPS %VBOASG %P 2:F139 = F327 + F139, 3: BOASG
         $FLAG[139] = $FLAG[327] OR $FLAG[139]
      ;ENDFOLD
      ;FOLD -- EZ2/SP2/KE2 oeffnen -- ;%{SE}%MKUKATPVW %CVW_COM %VCOMMENT %P 2:-- EZ2/SP2/KE2 oeffnen --, 3: VW_COMMENT
      ;ENDFOLD
      ;FOLD A878 = AUS ;%{SE}%MKUKATPVW %CVW_SPS %VBOASG %P 2:A878 = AUS, 3: BOASG
         $OUT[878] = FALSE
      ;ENDFOLD
      ;FOLD A877 = !E877 ;%{SE}%MKUKATPVW %CVW_SPS %VBOASG %P 2:A877 = !E877, 3: BOASG
         $OUT[877] = NOT $IN[877]
      ;ENDFOLD
      ;FOLD bin3 (F285) = 5 ;%{SE}%MKUKATPVW %CVW_SPS %VARIASG %P 2:bin3 (F285) = 5, 3: ARIASG
         VW(#BINOUT,$FLAG[285],3,5)
      ;ENDFOLD
      ;FOLD bin6 (!F285) = 1 ;%{SE}%MKUKATPVW %CVW_SPS %VARIASG %P 2:bin6 (!F285) = 1, 3: ARIASG
         VW(#BINOUT,NOT $FLAG[285],6,1)
      ;ENDFOLD
      ;FOLD -- Wartezeit Programmwechsel SK -- ;%{SE}%MKUKATPVW %CVW_COM %VCOMMENT %P 2:-- Wartezeit Programmwechsel SK --, 3: VW_COMMENT
      ;ENDFOLD
      ;FOLD T8 ( !F334 ) = -2[1/10Sek] ;%{SE}%MKUKATPVW %CVW_SPS %VTASG %P 2:T8 ( !F334 ) = -2[1/10Sek], 3: TASG
         VW(#SET_TIME,NOT $FLAG[334],8,0,-2)
      ;ENDFOLD
      ;FOLD -- Hilfsflag SK Programmwechsel -- ;%{SE}%MKUKATPVW %CVW_COM %VCOMMENT %P 2:-- Hilfsflag SK Programmwechsel --, 3: VW_COMMENT
      ;ENDFOLD
      ;FOLD F334 = EIN ;%{SE}%MKUKATPVW %CVW_SPS %VBOASG %P 2:F334 = EIN, 3: BOASG
         $FLAG[334] = TRUE
      ;ENDFOLD
      ;FOLD F748 = F322 + F323 + F325 + F326 + F327 + F329 ;%{SE}%MKUKATPVW %CVW_SPS %VBOASG %P 2:F748 = F322 + F323 + F325 + F326 + F327 + F329, 3: BOASG
         $FLAG[748] = $FLAG[322] OR $FLAG[323] OR $FLAG[325] OR $FLAG[326] OR $FLAG[327] OR $FLAG[329]
      ;ENDFOLD
      ;FOLD Schritt 74 = E877 & !E878 & (F322 + F323 + F325 + F326 + F327 + F329) & (E26 + E27) & A4039 ;%{SE}%MKUKATPVW %CVW_SPS %VST_CON %P 2:Schritt 74 = E877 & !E878 & (F322 + F323 + F325 + F326 + F327 + F329) & (E26 + E27) & A4039, 3: ST_CON
         IF $IN[877] AND NOT $IN[878] AND ($FLAG[322] OR $FLAG[323] OR $FLAG[325] OR $FLAG[326] OR $FLAG[327] OR $FLAG[329]) AND ($IN[26] OR $IN[27]) AND $OUT[4039] THEN
            PREVSTEP = $APP_INT[5]
            $APP_INT[5] = 74
         ENDIF
      ;ENDFOLD
      ;FOLD Schritt 74 = E877 & !E878 & (F322 + F323 + F325 + F326 + F327 + F329) & (F731 & F749) & A4039 ;%{SE}%MKUKATPVW %CVW_SPS %VST_CON %P 2:Schritt 74 = E877 & !E878 & (F322 + F323 + F325 + F326 + F327 + F329) & (F731 & F749) & A4039, 3: ST_CON
         IF $IN[877] AND NOT $IN[878] AND ($FLAG[322] OR $FLAG[323] OR $FLAG[325] OR $FLAG[326] OR $FLAG[327] OR $FLAG[329]) AND ($FLAG[731] AND $FLAG[749]) AND $OUT[4039] THEN
            PREVSTEP = $APP_INT[5]
            $APP_INT[5] = 74
         ENDIF
      ;ENDFOLD
      ;FOLD Schritt 96 = T8 & E877 & !E878 & (!F325 & !F326 & !F327 & !F329 + F160) & A4039 ;%{SE}%MKUKATPVW %CVW_SPS %VST_CON %P 2:Schritt 96 = T8 & E877 & !E878 & (!F325 & !F326 & !F327 & !F329 + F160) & A4039, 3: ST_CON
         IF $TIMER_FLAG[8] AND $IN[877] AND NOT $IN[878] AND (NOT $FLAG[325] AND NOT $FLAG[326] AND NOT $FLAG[327] AND NOT $FLAG[329] OR $FLAG[160]) AND $OUT[4039] THEN
            PREVSTEP = $APP_INT[5]
            $APP_INT[5] = 96
         ENDIF
      ;ENDFOLD
   ;ENDFOLD
   ;FOLD SCHRITT 96 -- STAT EZ2/SP2/KE2 # Ende -- ;%{P}%MKUKATPVW,%CSTEP,%VST_NR,%P 1:SCHRITT, 2:96, 3: STAT EZ2/SP2/KE2 # Ende
      ;FOLD ;%{H}
         Case 96
      ;ENDFOLD
      ;FOLD -- Hilfsflag SK Programmwechsel -- ;%{SE}%MKUKATPVW %CVW_COM %VCOMMENT %P 2:-- Hilfsflag SK Programmwechsel --, 3: VW_COMMENT
      ;ENDFOLD
      ;FOLD F334 = AUS ;%{SE}%MKUKATPVW %CVW_SPS %VBOASG %P 2:F334 = AUS, 3: BOASG
         $FLAG[334] = FALSE
      ;ENDFOLD
      ;FOLD -- RSK Sammelstoerung -- ;%{SE}%MKUKATPVW %CVW_COM %VCOMMENT %P 2:-- RSK Sammelstoerung --, 3: VW_COMMENT
      ;ENDFOLD
      ;FOLD F329 = F160 ;%{SE}%MKUKATPVW %CVW_SPS %VBOASG %P 2:F329 = F160, 3: BOASG
         $FLAG[329] = $FLAG[160]
      ;ENDFOLD
      ;FOLD F149 = (!F285 & !E946 & E947 &!E948 + F285 & !E786 & E787 & !E788) + F160 & (E26 + E27) ;%{SE}%MKUKATPVW %CVW_SPS %VBOASG %P 2:F149 = (!F285 & !E946 & E947 &!E948 + F285 & !E786 & E787 & !E788) + F160 & (E26 + E27), 3: BOASG
         $FLAG[149] = (NOT $FLAG[285] AND NOT $IN[946] AND $IN[947] AND NOT $IN[948] OR $FLAG[285] AND NOT $IN[786] AND $IN[787] AND NOT $IN[788]) OR $FLAG[160] AND ($IN[26] OR $IN[27])
      ;ENDFOLD
      ;FOLD Schritt 1 = F149 & A4039 ;%{SE}%MKUKATPVW %CVW_SPS %VST_CON %P 2:Schritt 1 = F149 & A4039, 3: ST_CON
         IF $FLAG[149] AND $OUT[4039] THEN
            PREVSTEP = $APP_INT[5]
            $APP_INT[5] = 1
         ENDIF
      ;ENDFOLD
   ;ENDFOLD
   ;FOLD SCHRITT 97 -- STAT EZ3/SP3/KE3 # Start -- ;%{P}%MKUKATPVW,%CSTEP,%VST_NR,%P 1:SCHRITT, 2:97, 3: STAT EZ3/SP3/KE3 # Start
      ;FOLD ;%{H}
         Case 97
      ;ENDFOLD
      ;FOLD -- RSK gestartet -- ;%{SE}%MKUKATPVW %CVW_COM %VCOMMENT %P 2:-- RSK gestartet --, 3: VW_COMMENT
      ;ENDFOLD
      ;FOLD F196 = AUS ;%{SE}%MKUKATPVW %CVW_SPS %VBOASG %P 2:F196 = AUS, 3: BOASG
         $FLAG[196] = FALSE
      ;ENDFOLD
      ;FOLD F321 = AUS ;%{SE}%MKUKATPVW %CVW_SPS %VBOASG %P 2:F321 = AUS, 3: BOASG
         $FLAG[321] = FALSE
      ;ENDFOLD
      ;FOLD F322 = AUS ;%{SE}%MKUKATPVW %CVW_SPS %VBOASG %P 2:F322 = AUS, 3: BOASG
         $FLAG[322] = FALSE
      ;ENDFOLD
      ;FOLD F323 = AUS ;%{SE}%MKUKATPVW %CVW_SPS %VBOASG %P 2:F323 = AUS, 3: BOASG
         $FLAG[323] = FALSE
      ;ENDFOLD
      ;FOLD F324 = AUS ;%{SE}%MKUKATPVW %CVW_SPS %VBOASG %P 2:F324 = AUS, 3: BOASG
         $FLAG[324] = FALSE
      ;ENDFOLD
      ;FOLD F325 = AUS ;%{SE}%MKUKATPVW %CVW_SPS %VBOASG %P 2:F325 = AUS, 3: BOASG
         $FLAG[325] = FALSE
      ;ENDFOLD
      ;FOLD F326 = AUS ;%{SE}%MKUKATPVW %CVW_SPS %VBOASG %P 2:F326 = AUS, 3: BOASG
         $FLAG[326] = FALSE
      ;ENDFOLD
      ;FOLD F327 = AUS ;%{SE}%MKUKATPVW %CVW_SPS %VBOASG %P 2:F327 = AUS, 3: BOASG
         $FLAG[327] = FALSE
      ;ENDFOLD
      ;FOLD F329 = AUS ;%{SE}%MKUKATPVW %CVW_SPS %VBOASG %P 2:F329 = AUS, 3: BOASG
         $FLAG[329] = FALSE
      ;ENDFOLD
      ;FOLD -- EZ3/SP3/KE3 Zaehler -- ;%{SE}%MKUKATPVW %CVW_COM %VCOMMENT %P 2:-- EZ3/SP3/KE3 Zaehler --, 3: VW_COMMENT
      ;ENDFOLD
      ;FOLD F186 = AUS ;%{SE}%MKUKATPVW %CVW_SPS %VBOASG %P 2:F186 = AUS, 3: BOASG
         $FLAG[186] = FALSE
      ;ENDFOLD
      ;FOLD F187 = AUS ;%{SE}%MKUKATPVW %CVW_SPS %VBOASG %P 2:F187 = AUS, 3: BOASG
         $FLAG[187] = FALSE
      ;ENDFOLD
      ;FOLD F188 = AUS ;%{SE}%MKUKATPVW %CVW_SPS %VBOASG %P 2:F188 = AUS, 3: BOASG
         $FLAG[188] = FALSE
      ;ENDFOLD
      ;FOLD F189 = AUS ;%{SE}%MKUKATPVW %CVW_SPS %VBOASG %P 2:F189 = AUS, 3: BOASG
         $FLAG[189] = FALSE
      ;ENDFOLD
      ;FOLD F190 = AUS ;%{SE}%MKUKATPVW %CVW_SPS %VBOASG %P 2:F190 = AUS, 3: BOASG
         $FLAG[190] = FALSE
      ;ENDFOLD
      ;FOLD F191 = AUS ;%{SE}%MKUKATPVW %CVW_SPS %VBOASG %P 2:F191 = AUS, 3: BOASG
         $FLAG[191] = FALSE
      ;ENDFOLD
      ;FOLD -- Hilfsflags Funktionstest KF Motor -- ;%{SE}%MKUKATPVW %CVW_COM %VCOMMENT %P 2:-- Hilfsflags Funktionstest KF Motor --, 3: VW_COMMENT
      ;ENDFOLD
      ;FOLD F312 = AUS ;%{SE}%MKUKATPVW %CVW_SPS %VBOASG %P 2:F312 = AUS, 3: BOASG
         $FLAG[312] = FALSE
      ;ENDFOLD
      ;FOLD F313 = AUS ;%{SE}%MKUKATPVW %CVW_SPS %VBOASG %P 2:F313 = AUS, 3: BOASG
         $FLAG[313] = FALSE
      ;ENDFOLD
      ;FOLD bin7 ( !F832 ) = 31 ;%{SE}%MKUKATPVW %CVW_SPS %VARIASG %P 2:bin7 ( !F832 ) = 31, 3: ARIASG
         VW(#BINOUT,NOT $FLAG[832],7,31)
      ;ENDFOLD
      ;FOLD bin9 ( EIN ) = 31 ;%{SE}%MKUKATPVW %CVW_SPS %VARIASG %P 2:bin9 ( EIN ) = 31, 3: ARIASG
         VW(#BINOUT,TRUE,9,31)
      ;ENDFOLD
      ;FOLD -- Wartezeit Programmwechsel SK -- ;%{SE}%MKUKATPVW %CVW_COM %VCOMMENT %P 2:-- Wartezeit Programmwechsel SK --, 3: VW_COMMENT
      ;ENDFOLD
      ;FOLD T8 ( !F334 ) = -2[1/10Sek] ;%{SE}%MKUKATPVW %CVW_SPS %VTASG %P 2:T8 ( !F334 ) = -2[1/10Sek], 3: TASG
         VW(#SET_TIME,NOT $FLAG[334],8,0,-2)
      ;ENDFOLD
      ;FOLD -- Hilfsflag SK Programmwechsel -- ;%{SE}%MKUKATPVW %CVW_COM %VCOMMENT %P 2:-- Hilfsflag SK Programmwechsel --, 3: VW_COMMENT
      ;ENDFOLD
      ;FOLD F334 = EIN ;%{SE}%MKUKATPVW %CVW_SPS %VBOASG %P 2:F334 = EIN, 3: BOASG
         $FLAG[334] = TRUE
      ;ENDFOLD
      ;FOLD -- Quitt. Fraesen SK3 AUS -- ;%{SE}%MKUKATPVW %CVW_COM %VCOMMENT %P 2:-- Quitt. Fraesen SK3 AUS --, 3: VW_COMMENT
      ;ENDFOLD
      ;FOLD A1106 = AUS ;%{SE}%MKUKATPVW %CVW_SPS %VBOASG %P 2:A1106 = AUS, 3: BOASG
         $OUT[1106] = FALSE
      ;ENDFOLD
      ;FOLD Schritt 98 = T8 & A4039 ;%{SE}%MKUKATPVW %CVW_SPS %VST_CON %P 2:Schritt 98 = T8 & A4039, 3: ST_CON
         IF $TIMER_FLAG[8] AND $OUT[4039] THEN
            PREVSTEP = $APP_INT[5]
            $APP_INT[5] = 98
         ENDIF
      ;ENDFOLD
   ;ENDFOLD
   ;FOLD SCHRITT 98 -- STAT EZ3/SP3/KE3 -- ;%{P}%MKUKATPVW,%CSTEP,%VST_NR,%P 1:SCHRITT, 2:98, 3: STAT EZ3/SP3/KE3
      ;FOLD ;%{H}
         Case 98
      ;ENDFOLD
      ;FOLD -- Fraeszyklen fuer autom. KF-Umderhung -- ;%{SE}%MKUKATPVW %CVW_COM %VCOMMENT %P 2:-- Fraeszyklen fuer autom. KF-Umderhung --, 3: VW_COMMENT
      ;ENDFOLD
      ;FOLD i36 (EIN) = i36 + 1 ;%{SE}%MKUKATPVW %CVW_SPS %VARIASG %P 2:i36 (EIN) = i36 + 1, 3: ARIASG
         VW(#COUNTER,TRUE,36,$COUNT_I[36] + 1)
      ;ENDFOLD
      ;FOLD -- Hilfsflag SK Programmwechsel -- ;%{SE}%MKUKATPVW %CVW_COM %VCOMMENT %P 2:-- Hilfsflag SK Programmwechsel --, 3: VW_COMMENT
      ;ENDFOLD
      ;FOLD F334 = AUS ;%{SE}%MKUKATPVW %CVW_SPS %VBOASG %P 2:F334 = AUS, 3: BOASG
         $FLAG[334] = FALSE
      ;ENDFOLD
      ;FOLD -- Ueberwachungszeit KF3 EIN -- ;%{SE}%MKUKATPVW %CVW_COM %VCOMMENT %P 2:-- Ueberwachungszeit KF3 EIN --, 3: VW_COMMENT
      ;ENDFOLD
      ;FOLD T7 ( EIN ) = -30[1/10Sek] ;%{SE}%MKUKATPVW %CVW_SPS %VTASG %P 2:T7 ( EIN ) = -30[1/10Sek], 3: TASG
         VW(#SET_TIME,TRUE,7,0,-30)
      ;ENDFOLD
      ;FOLD -- KF3 einschalten -- ;%{SE}%MKUKATPVW %CVW_COM %VCOMMENT %P 2:-- KF3 einschalten --, 3: VW_COMMENT
      ;ENDFOLD
      ;FOLD i1 (EIN) = 0 ;%{SE}%MKUKATPVW %CVW_SPS %VARIASG %P 2:i1 (EIN) = 0, 3: ARIASG
         VW(#COUNTER,TRUE,1,0)
      ;ENDFOLD
      ;FOLD A1154 = EIN ;%{SE}%MKUKATPVW %CVW_SPS %VBOASG %P 2:A1154 = EIN, 3: BOASG
         $OUT[1154] = TRUE
      ;ENDFOLD
      ;FOLD Schritt 99 = A4039 ;%{SE}%MKUKATPVW %CVW_SPS %VST_CON %P 2:Schritt 99 = A4039, 3: ST_CON
         IF $OUT[4039] THEN
            PREVSTEP = $APP_INT[5]
            $APP_INT[5] = 99
         ENDIF
      ;ENDFOLD
   ;ENDFOLD
   ;FOLD SCHRITT 99 -- STAT EZ3/SP3/KE3 -- ;%{P}%MKUKATPVW,%CSTEP,%VST_NR,%P 1:SCHRITT, 2:99, 3: STAT EZ3/SP3/KE3
      ;FOLD ;%{H}
         Case 99
      ;ENDFOLD
      ;FOLD -- Funktionstest KF Motor -- ;%{SE}%MKUKATPVW %CVW_COM %VCOMMENT %P 2:-- Funktionstest KF Motor --, 3: VW_COMMENT
      ;ENDFOLD
      ;FOLD F312 = EIN ;%{SE}%MKUKATPVW %CVW_SPS %VBOASG %P 2:F312 = EIN, 3: BOASG
         $FLAG[312] = TRUE
      ;ENDFOLD
      ;FOLD F313 = i1 > 2 ;%{SE}%MKUKATPVW %CVW_SPS %VBOCMP %P 2:F313 = i1 > 2, 3: BOCMP
         $FLAG[313] = $COUNT_I[1] > 2
      ;ENDFOLD
      ;FOLD Schritt 100 = (F313 + T7) & A4039 ;%{SE}%MKUKATPVW %CVW_SPS %VST_CON %P 2:Schritt 100 = (F313 + T7) & A4039, 3: ST_CON
         IF ($FLAG[313] OR $TIMER_FLAG[7]) AND $OUT[4039] THEN
            PREVSTEP = $APP_INT[5]
            $APP_INT[5] = 100
         ENDIF
      ;ENDFOLD
   ;ENDFOLD
   ;FOLD SCHRITT 100 -- STAT EZ3/SP3/KE3 -- ;%{P}%MKUKATPVW,%CSTEP,%VST_NR,%P 1:SCHRITT, 2:100, 3: STAT EZ3/SP3/KE3
      ;FOLD ;%{H}
         Case 100
      ;ENDFOLD
      ;FOLD F312 = AUS ;%{SE}%MKUKATPVW %CVW_SPS %VBOASG %P 2:F312 = AUS, 3: BOASG
         $FLAG[312] = FALSE
      ;ENDFOLD
      ;FOLD -- Ueberwachungszeit KS3 schwenken -- ;%{SE}%MKUKATPVW %CVW_COM %VCOMMENT %P 2:-- Ueberwachungszeit KS3 schwenken --, 3: VW_COMMENT
      ;ENDFOLD
      ;FOLD t8 ( EIN ) = -100[1/10Sek] ;%{SE}%MKUKATPVW %CVW_SPS %VTASG %P 2:t8 ( EIN ) = -100[1/10Sek], 3: TASG
         VW(#SET_TIME,TRUE,8,0,-100)
      ;ENDFOLD
      ;FOLD Schritt 101 = A4039 ;%{SE}%MKUKATPVW %CVW_SPS %VST_CON %P 2:Schritt 101 = A4039, 3: ST_CON
         IF $OUT[4039] THEN
            PREVSTEP = $APP_INT[5]
            $APP_INT[5] = 101
         ENDIF
      ;ENDFOLD
   ;ENDFOLD
   ;FOLD SCHRITT 101 -- STAT EZ3/SP3/KE3 -- ;%{P}%MKUKATPVW,%CSTEP,%VST_NR,%P 1:SCHRITT, 2:101, 3: STAT EZ3/SP3/KE3
      ;FOLD ;%{H}
         Case 101
      ;ENDFOLD
      ;FOLD -- RSK Fehlerausgabe KF1 Initiator/Motor -- ;%{SE}%MKUKATPVW %CVW_COM %VCOMMENT %P 2:-- RSK Fehlerausgabe KF1 Initiator/Motor --, 3: VW_COMMENT
      ;ENDFOLD
      ;FOLD F322 = !F313 ;%{SE}%MKUKATPVW %CVW_SPS %VBOASG %P 2:F322 = !F313, 3: BOASG
         $FLAG[322] = NOT $FLAG[313]
      ;ENDFOLD
      ;FOLD -- RSK Fehlerausgabe KS3 Ruhest. -- ;%{SE}%MKUKATPVW %CVW_COM %VCOMMENT %P 2:-- RSK Fehlerausgabe KS3 Ruhest. --, 3: VW_COMMENT
      ;ENDFOLD
      ;FOLD F323 = (!E1156 + E1157 + E1158 + !E1159) & !F324 & !F328 ;%{SE}%MKUKATPVW %CVW_SPS %VBOASG %P 2:F323 = (!E1156 + E1157 + E1158 + !E1159) & !F324 & !F328, 3: BOASG
         $FLAG[323] = (NOT $IN[1156] OR $IN[1157] OR $IN[1158] OR NOT $IN[1159]) AND NOT $FLAG[324] AND NOT $FLAG[328]
      ;ENDFOLD
      ;FOLD -- RSK Sammelstoerung -- ;%{SE}%MKUKATPVW %CVW_COM %VCOMMENT %P 2:-- RSK Sammelstoerung --, 3: VW_COMMENT
      ;ENDFOLD
      ;FOLD F329 = F322 + F323 ;%{SE}%MKUKATPVW %CVW_SPS %VBOASG %P 2:F329 = F322 + F323, 3: BOASG
         $FLAG[329] = $FLAG[322] OR $FLAG[323]
      ;ENDFOLD
      ;FOLD T7 ( EIN ) = STOP ;%{SE}%MKUKATPVW %CVW_SPS %VTSTOP %P 2:T7 ( EIN ) = STOP, 3: TSTOP
         VW(#SET_TIME,TRUE,7,1,0)
      ;ENDFOLD
      ;FOLD A1154 = !F322 & !F323 ;%{SE}%MKUKATPVW %CVW_SPS %VBOASG %P 2:A1154 = !F322 & !F323, 3: BOASG
         $OUT[1154] = NOT $FLAG[322] AND NOT $FLAG[323]
      ;ENDFOLD
      ;FOLD -- KF3 Versetzeinheit vor -- ;%{SE}%MKUKATPVW %CVW_COM %VCOMMENT %P 2:-- KF3 Versetzeinheit vor --, 3: VW_COMMENT
      ;ENDFOLD
      ;FOLD A1155 = !F322 & !F323 & F566 ;%{SE}%MKUKATPVW %CVW_SPS %VBOASG %P 2:A1155 = !F322 & !F323 & F566, 3: BOASG
         $OUT[1155] = NOT $FLAG[322] AND NOT $FLAG[323] AND $FLAG[566]
      ;ENDFOLD
      ;FOLD Schritt 102 = (!F322 & !F323 & (E1155 & F566 + !E1155 & !F566) + T8) & A4039 ;%{SE}%MKUKATPVW %CVW_SPS %VST_CON %P 2:Schritt 102 = (!F322 & !F323 & (E1155 & F566 + !E1155 & !F566) + T8) & A4039, 3: ST_CON
         IF (NOT $FLAG[322] AND NOT $FLAG[323] AND ($IN[1155] AND $FLAG[566] OR NOT $IN[1155] AND NOT $FLAG[566]) OR $TIMER_FLAG[8]) AND $OUT[4039] THEN
            PREVSTEP = $APP_INT[5]
            $APP_INT[5] = 102
         ENDIF
      ;ENDFOLD
      ;FOLD Schritt 118 = (F322 + F323) & !F324 & !F328 & A4039 ;%{SE}%MKUKATPVW %CVW_SPS %VST_CON %P 2:Schritt 118 = (F322 + F323) & !F324 & !F328 & A4039, 3: ST_CON
         IF ($FLAG[322] OR $FLAG[323]) AND NOT $FLAG[324] AND NOT $FLAG[328] AND $OUT[4039] THEN
            PREVSTEP = $APP_INT[5]
            $APP_INT[5] = 118
         ENDIF
      ;ENDFOLD
   ;ENDFOLD
   ;FOLD SCHRITT 102 -- STAT EZ3/SP3/KE3 -- ;%{P}%MKUKATPVW,%CSTEP,%VST_NR,%P 1:SCHRITT, 2:102, 3: STAT EZ3/SP3/KE3
      ;FOLD ;%{H}
         Case 102
      ;ENDFOLD
      ;FOLD F329 = T8 ;%{SE}%MKUKATPVW %CVW_SPS %VBOASG %P 2:F329 = T8, 3: BOASG
         $FLAG[329] = $TIMER_FLAG[8]
      ;ENDFOLD
      ;FOLD F324 = AUS ;%{SE}%MKUKATPVW %CVW_SPS %VBOASG %P 2:F324 = AUS, 3: BOASG
         $FLAG[324] = FALSE
      ;ENDFOLD
      ;FOLD F328 = AUS ;%{SE}%MKUKATPVW %CVW_SPS %VBOASG %P 2:F328 = AUS, 3: BOASG
         $FLAG[328] = FALSE
      ;ENDFOLD
      ;FOLD -- KS3 in Arbeitsstellung schwenken -- ;%{SE}%MKUKATPVW %CVW_COM %VCOMMENT %P 2:-- KS3 in Arbeitsstellung schwenken --, 3: VW_COMMENT
      ;ENDFOLD
      ;FOLD A1160 = (F747 + !F714) & E1037 & !E1157 & (E1155 & F566 + !E1155 & !F566) ;%{SE}%MKUKATPVW %CVW_SPS %VBOASG %P 2:A1160 = (F747 + !F714) & E1037 & !E1157 & (E1155 & F566 + !E1155 & !F566), 3: BOASG
         $OUT[1160] = ($FLAG[747] OR NOT $FLAG[714]) AND $IN[1037] AND NOT $IN[1157] AND ($IN[1155] AND $FLAG[566] OR NOT $IN[1155] AND NOT $FLAG[566])
      ;ENDFOLD
      ;FOLD -- KF3 Ausblasen -- ;%{SE}%MKUKATPVW %CVW_COM %VCOMMENT %P 2:-- KF3 Ausblasen --, 3: VW_COMMENT
      ;ENDFOLD
      ;FOLD A1156 = F330 + !F330 & !F331 & !F332 ;%{SE}%MKUKATPVW %CVW_SPS %VBOASG %P 2:A1156 = F330 + !F330 & !F331 & !F332, 3: BOASG
         $OUT[1156] = $FLAG[330] OR NOT $FLAG[330] AND NOT $FLAG[331] AND NOT $FLAG[332]
      ;ENDFOLD
      ;FOLD Schritt 103 = (F747 + !F714) & E1037 & (A1160 + E1157 + T8) & A4039 ;%{SE}%MKUKATPVW %CVW_SPS %VST_CON %P 2:Schritt 103 = (F747 + !F714) & E1037 & (A1160 + E1157 + T8) & A4039, 3: ST_CON
         IF ($FLAG[747] OR NOT $FLAG[714]) AND $IN[1037] AND ($OUT[1160] OR $IN[1157] OR $TIMER_FLAG[8]) AND $OUT[4039] THEN
            PREVSTEP = $APP_INT[5]
            $APP_INT[5] = 103
         ENDIF
      ;ENDFOLD
   ;ENDFOLD
   ;FOLD SCHRITT 103 -- STAT EZ3/SP3/KE3 -- ;%{P}%MKUKATPVW,%CSTEP,%VST_NR,%P 1:SCHRITT, 2:103, 3: STAT EZ3/SP3/KE3
      ;FOLD ;%{H}
         Case 103
      ;ENDFOLD
      ;FOLD -- RSK Fehlerausgabe KF Versetzeinheit -- ;%{SE}%MKUKATPVW %CVW_COM %VCOMMENT %P 2:-- RSK Fehlerausgabe KF Versetzeinheit --, 3: VW_COMMENT
      ;ENDFOLD
      ;FOLD F328 = !E1155 & F566 & !F324 ;%{SE}%MKUKATPVW %CVW_SPS %VBOASG %P 2:F328 = !E1155 & F566 & !F324, 3: BOASG
         $FLAG[328] = NOT $IN[1155] AND $FLAG[566] AND NOT $FLAG[324]
      ;ENDFOLD
      ;FOLD -- RSK Fehlerausgabe KS3 Arbeitsstellung -- ;%{SE}%MKUKATPVW %CVW_COM %VCOMMENT %P 2:-- RSK Fehlerausgabe KS3 Arbeitsstellung --, 3: VW_COMMENT
      ;ENDFOLD
      ;FOLD F324 = (E1156 + !E1157 + !E1158 + E1159) & T8 & (E1155 + !F566) + F324 ;%{SE}%MKUKATPVW %CVW_SPS %VBOASG %P 2:F324 = (E1156 + !E1157 + !E1158 + E1159) & T8 & (E1155 + !F566) + F324, 3: BOASG
         $FLAG[324] = ($IN[1156] OR NOT $IN[1157] OR NOT $IN[1158] OR $IN[1159]) AND $TIMER_FLAG[8] AND ($IN[1155] OR NOT $FLAG[566]) OR $FLAG[324]
      ;ENDFOLD
      ;FOLD -- RSK Fehlerausgabe EZ/SP min. Oeffnung -- ;%{SE}%MKUKATPVW %CVW_COM %VCOMMENT %P 2:-- RSK Fehlerausgabe EZ/SP min. Oeffnung --, 3: VW_COMMENT
      ;ENDFOLD
      ;FOLD F333 = !F747 ;%{SE}%MKUKATPVW %CVW_SPS %VBOASG %P 2:F333 = !F747, 3: BOASG
         $FLAG[333] = NOT $FLAG[747]
      ;ENDFOLD
      ;FOLD -- RSK Sammelstoerung -- ;%{SE}%MKUKATPVW %CVW_COM %VCOMMENT %P 2:-- RSK Sammelstoerung --, 3: VW_COMMENT
      ;ENDFOLD
      ;FOLD F329 = F324 + F328 ;%{SE}%MKUKATPVW %CVW_SPS %VBOASG %P 2:F329 = F324 + F328, 3: BOASG
         $FLAG[329] = $FLAG[324] OR $FLAG[328]
      ;ENDFOLD
      ;FOLD A1154 = !F324 & !F328 ;%{SE}%MKUKATPVW %CVW_SPS %VBOASG %P 2:A1154 = !F324 & !F328, 3: BOASG
         $OUT[1154] = NOT $FLAG[324] AND NOT $FLAG[328]
      ;ENDFOLD
      ;FOLD -- KF3 Ausblasen -- ;%{SE}%MKUKATPVW %CVW_COM %VCOMMENT %P 2:-- KF3 Ausblasen --, 3: VW_COMMENT
      ;ENDFOLD
      ;FOLD A1156 = (F330 + !F330 & !F331 & !F332) & !F324 & !F328 ;%{SE}%MKUKATPVW %CVW_SPS %VBOASG %P 2:A1156 = (F330 + !F330 & !F331 & !F332) & !F324 & !F328, 3: BOASG
         $OUT[1156] = ($FLAG[330] OR NOT $FLAG[330] AND NOT $FLAG[331] AND NOT $FLAG[332]) AND NOT $FLAG[324] AND NOT $FLAG[328]
      ;ENDFOLD
      ;FOLD A1155 = F566 ;%{SE}%MKUKATPVW %CVW_SPS %VBOASG %P 2:A1155 = F566, 3: BOASG
         $OUT[1155] = $FLAG[566]
      ;ENDFOLD
      ;FOLD -- Ueberwachungszeit EZ3/SP3/KE3 schliessen -- ;%{SE}%MKUKATPVW %CVW_COM %VCOMMENT %P 2:-- Ueberwachungszeit EZ3/SP3/KE3 schliessen --, 3: VW_COMMENT
      ;ENDFOLD
      ;FOLD t9 ( EIN ) = -100[1/10Sek] ;%{SE}%MKUKATPVW %CVW_SPS %VTASG %P 2:t9 ( EIN ) = -100[1/10Sek], 3: TASG
         VW(#SET_TIME,TRUE,9,0,-100)
      ;ENDFOLD
      ;FOLD -- Verweilzeit Versetzeinheit Rueck -- ;%{SE}%MKUKATPVW %CVW_COM %VCOMMENT %P 2:-- Verweilzeit Versetzeinheit Rueck --, 3: VW_COMMENT
      ;ENDFOLD
      ;FOLD t11 ( EIN ) = i24[1/10Sek] ;%{SE}%MKUKATPVW %CVW_SPS %VTASG %P 2:t11 ( EIN ) = i24[1/10Sek], 3: TASG
         VW(#SET_TIME,TRUE,11,0,$COUNT_I[24])
      ;ENDFOLD
      ;FOLD Schritt 98 = (F324 + F328) & (E26 + E27) & A4039 ;%{SE}%MKUKATPVW %CVW_SPS %VST_CON %P 2:Schritt 98 = (F324 + F328) & (E26 + E27) & A4039, 3: ST_CON
         IF ($FLAG[324] OR $FLAG[328]) AND ($IN[26] OR $IN[27]) AND $OUT[4039] THEN
            PREVSTEP = $APP_INT[5]
            $APP_INT[5] = 98
         ENDIF
      ;ENDFOLD
      ;FOLD Schritt 104 = !F324 & !F328 & !E1156 & E1157 & E1158 & !E1159 & A4039 ;%{SE}%MKUKATPVW %CVW_SPS %VST_CON %P 2:Schritt 104 = !F324 & !F328 & !E1156 & E1157 & E1158 & !E1159 & A4039, 3: ST_CON
         IF NOT $FLAG[324] AND NOT $FLAG[328] AND NOT $IN[1156] AND $IN[1157] AND $IN[1158] AND NOT $IN[1159] AND $OUT[4039] THEN
            PREVSTEP = $APP_INT[5]
            $APP_INT[5] = 104
         ENDIF
      ;ENDFOLD
   ;ENDFOLD
   ;FOLD SCHRITT 104 -- STAT EZ3/SP3/KE3 -- ;%{P}%MKUKATPVW,%CSTEP,%VST_NR,%P 1:SCHRITT, 2:104, 3: STAT EZ3/SP3/KE3
      ;FOLD ;%{H}
         Case 104
      ;ENDFOLD
      ;FOLD -- Umdreh. KF setzen zwischenspeichern -- ;%{SE}%MKUKATPVW %CVW_COM %VCOMMENT %P 2:-- Umdreh. KF setzen zwischenspeichern --, 3: VW_COMMENT
      ;ENDFOLD
      ;FOLD i45 ( EIN ) = i19 ;%{SE}%MKUKATPVW %CVW_SPS %VARIASG %P 2:i45 ( EIN ) = i19, 3: ARIASG
         VW(#COUNTER,TRUE,45,$COUNT_I[19])
      ;ENDFOLD
      ;FOLD i19 ( F155 ) = i44 ;%{SE}%MKUKATPVW %CVW_SPS %VARIASG %P 2:i19 ( F155 ) = i44, 3: ARIASG
         VW(#COUNTER,$FLAG[155],19,$COUNT_I[44])
      ;ENDFOLD
      ;FOLD i1 ( EIN ) = 0 ;%{SE}%MKUKATPVW %CVW_SPS %VARIASG %P 2:i1 ( EIN ) = 0, 3: ARIASG
         VW(#COUNTER,TRUE,1,0)
      ;ENDFOLD
      ;FOLD F190 = AUS ;%{SE}%MKUKATPVW %CVW_SPS %VBOASG %P 2:F190 = AUS, 3: BOASG
         $FLAG[190] = FALSE
      ;ENDFOLD
      ;FOLD F312 = AUS ;%{SE}%MKUKATPVW %CVW_SPS %VBOASG %P 2:F312 = AUS, 3: BOASG
         $FLAG[312] = FALSE
      ;ENDFOLD
      ;FOLD F313 = AUS ;%{SE}%MKUKATPVW %CVW_SPS %VBOASG %P 2:F313 = AUS, 3: BOASG
         $FLAG[313] = FALSE
      ;ENDFOLD
      ;FOLD F324 = AUS ;%{SE}%MKUKATPVW %CVW_SPS %VBOASG %P 2:F324 = AUS, 3: BOASG
         $FLAG[324] = FALSE
      ;ENDFOLD
      ;FOLD F328 = AUS ;%{SE}%MKUKATPVW %CVW_SPS %VBOASG %P 2:F328 = AUS, 3: BOASG
         $FLAG[328] = FALSE
      ;ENDFOLD
      ;FOLD -- KF3 einschalten nach Fehler -- ;%{SE}%MKUKATPVW %CVW_COM %VCOMMENT %P 2:-- KF3 einschalten nach Fehler --, 3: VW_COMMENT
      ;ENDFOLD
      ;FOLD A1154 = EIN ;%{SE}%MKUKATPVW %CVW_SPS %VBOASG %P 2:A1154 = EIN, 3: BOASG
         $OUT[1154] = TRUE
      ;ENDFOLD
      ;FOLD -- KF3 Versetzeinheit rueck -- ;%{SE}%MKUKATPVW %CVW_COM %VCOMMENT %P 2:-- KF3 Versetzeinheit rueck --, 3: VW_COMMENT
      ;ENDFOLD
      ;FOLD A1155 = AUS ;%{SE}%MKUKATPVW %CVW_SPS %VBOASG %P 2:A1155 = AUS, 3: BOASG
         $OUT[1155] = FALSE
      ;ENDFOLD
      ;FOLD Schritt 105 = T11 & A4039 ;%{SE}%MKUKATPVW %CVW_SPS %VST_CON %P 2:Schritt 105 = T11 & A4039, 3: ST_CON
         IF $TIMER_FLAG[11] AND $OUT[4039] THEN
            PREVSTEP = $APP_INT[5]
            $APP_INT[5] = 105
         ENDIF
      ;ENDFOLD
   ;ENDFOLD
   ;FOLD SCHRITT 105 -- STAT EZ3/SP3/KE3 -- ;%{P}%MKUKATPVW,%CSTEP,%VST_NR,%P 1:SCHRITT, 2:105, 3: STAT EZ3/SP3/KE3
      ;FOLD ;%{H}
         Case 105
      ;ENDFOLD
      ;FOLD t11 ( EIN ) = STOP ;%{SE}%MKUKATPVW %CVW_SPS %VTSTOP %P 2:t11 ( EIN ) = STOP, 3: TSTOP
         VW(#SET_TIME,TRUE,11,1,0)
      ;ENDFOLD
      ;FOLD -- EZ3/SP3/KE3 schliessen -- ;%{SE}%MKUKATPVW %CVW_COM %VCOMMENT %P 2:-- EZ3/SP3/KE3 schliessen --, 3: VW_COMMENT
      ;ENDFOLD
      ;FOLD A1037 = AUS ;%{SE}%MKUKATPVW %CVW_SPS %VBOASG %P 2:A1037 = AUS, 3: BOASG
         $OUT[1037] = FALSE
      ;ENDFOLD
      ;FOLD -- EZ3/SP3 -- ;%{SE}%MKUKATPVW %CVW_COM %VCOMMENT %P 2:-- EZ3/SP3 --, 3: VW_COMMENT
      ;ENDFOLD
      ;FOLD A1038 = !F832 ;%{SE}%MKUKATPVW %CVW_SPS %VBOASG %P 2:A1038 = !F832, 3: BOASG
         $OUT[1038] = NOT $FLAG[832]
      ;ENDFOLD
      ;FOLD -- KE3 -- ;%{SE}%MKUKATPVW %CVW_COM %VCOMMENT %P 2:-- KE3 --, 3: VW_COMMENT
      ;ENDFOLD
      ;FOLD A1086 = F832 ;%{SE}%MKUKATPVW %CVW_SPS %VBOASG %P 2:A1086 = F832, 3: BOASG
         $OUT[1086] = $FLAG[832]
      ;ENDFOLD
      ;FOLD -- KF3 Ausblasen -- ;%{SE}%MKUKATPVW %CVW_COM %VCOMMENT %P 2:-- KF3 Ausblasen --, 3: VW_COMMENT
      ;ENDFOLD
      ;FOLD A1156 = F330 + F331 + !F330 & !F331 & !F332 ;%{SE}%MKUKATPVW %CVW_SPS %VBOASG %P 2:A1156 = F330 + F331 + !F330 & !F331 & !F332, 3: BOASG
         $OUT[1156] = $FLAG[330] OR $FLAG[331] OR NOT $FLAG[330] AND NOT $FLAG[331] AND NOT $FLAG[332]
      ;ENDFOLD
      ;FOLD Schritt 106 = (!E1037 & E1038 + T9) & A4039 ;%{SE}%MKUKATPVW %CVW_SPS %VST_CON %P 2:Schritt 106 = (!E1037 & E1038 + T9) & A4039, 3: ST_CON
         IF (NOT $IN[1037] AND $IN[1038] OR $TIMER_FLAG[9]) AND $OUT[4039] THEN
            PREVSTEP = $APP_INT[5]
            $APP_INT[5] = 106
         ENDIF
      ;ENDFOLD
   ;ENDFOLD
   ;FOLD SCHRITT 106 -- STAT EZ3/SP3/KE3 -- ;%{P}%MKUKATPVW,%CSTEP,%VST_NR,%P 1:SCHRITT, 2:106, 3: STAT EZ3/SP3/KE3
      ;FOLD ;%{H}
         Case 106
      ;ENDFOLD
      ;FOLD -- RSK Fehlerausgabe Kraftaufbau -- ;%{SE}%MKUKATPVW %CVW_COM %VCOMMENT %P 2:-- RSK Fehlerausgabe Kraftaufbau --, 3: VW_COMMENT
      ;ENDFOLD
      ;FOLD F325 = T9 ;%{SE}%MKUKATPVW %CVW_SPS %VBOASG %P 2:F325 = T9, 3: BOASG
         $FLAG[325] = $TIMER_FLAG[9]
      ;ENDFOLD
      ;FOLD -- RSK Sammelstoerung -- ;%{SE}%MKUKATPVW %CVW_COM %VCOMMENT %P 2:-- RSK Sammelstoerung --, 3: VW_COMMENT
      ;ENDFOLD
      ;FOLD F329 = F325 ;%{SE}%MKUKATPVW %CVW_SPS %VBOASG %P 2:F329 = F325, 3: BOASG
         $FLAG[329] = $FLAG[325]
      ;ENDFOLD
      ;FOLD -- KF3 abschalten bei Fehler -- ;%{SE}%MKUKATPVW %CVW_COM %VCOMMENT %P 2:-- KF3 abschalten bei Fehler --, 3: VW_COMMENT
      ;ENDFOLD
      ;FOLD A1154 = !T9 ;%{SE}%MKUKATPVW %CVW_SPS %VBOASG %P 2:A1154 = !T9, 3: BOASG
         $OUT[1154] = NOT $TIMER_FLAG[9]
      ;ENDFOLD
      ;FOLD -- KF3 Ausblasen -- ;%{SE}%MKUKATPVW %CVW_COM %VCOMMENT %P 2:-- KF3 Ausblasen --, 3: VW_COMMENT
      ;ENDFOLD
      ;FOLD A1156 = (F330 + F331 + !F330 & !F331 & !F332) & !T9 ;%{SE}%MKUKATPVW %CVW_SPS %VBOASG %P 2:A1156 = (F330 + F331 + !F330 & !F331 & !F332) & !T9, 3: BOASG
         $OUT[1156] = ($FLAG[330] OR $FLAG[331] OR NOT $FLAG[330] AND NOT $FLAG[331] AND NOT $FLAG[332]) AND NOT $TIMER_FLAG[9]
      ;ENDFOLD
      ;FOLD -- Warte Fraesen fertig oder Timeout -- ;%{SE}%MKUKATPVW %CVW_COM %VCOMMENT %P 2:-- Warte Fraesen fertig oder Timeout --, 3: VW_COMMENT
      ;ENDFOLD
      ;FOLD Schritt 107 = (F175 & F190 + F174 & F186 & !F287 + T7 + T9 + F325) & A4039 ;%{SE}%MKUKATPVW %CVW_SPS %VST_CON %P 2:Schritt 107 = (F175 & F190 + F174 & F186 & !F287 + T7 + T9 + F325) & A4039, 3: ST_CON
         IF ($FLAG[175] AND $FLAG[190] OR $FLAG[174] AND $FLAG[186] AND NOT $FLAG[287] OR $TIMER_FLAG[7] OR $TIMER_FLAG[9] OR $FLAG[325]) AND $OUT[4039] THEN
            PREVSTEP = $APP_INT[5]
            $APP_INT[5] = 107
         ENDIF
      ;ENDFOLD
      ;FOLD Schritt 107 = (F174 & F188 & F287 + T7 + T9 + F325) & A4039 ;%{SE}%MKUKATPVW %CVW_SPS %VST_CON %P 2:Schritt 107 = (F174 & F188 & F287 + T7 + T9 + F325) & A4039, 3: ST_CON
         IF ($FLAG[174] AND $FLAG[188] AND $FLAG[287] OR $TIMER_FLAG[7] OR $TIMER_FLAG[9] OR $FLAG[325]) AND $OUT[4039] THEN
            PREVSTEP = $APP_INT[5]
            $APP_INT[5] = 107
         ENDIF
      ;ENDFOLD
   ;ENDFOLD
   ;FOLD SCHRITT 107 -- STAT EZ3/SP3/KE3 -- ;%{P}%MKUKATPVW,%CSTEP,%VST_NR,%P 1:SCHRITT, 2:107, 3: STAT EZ3/SP3/KE3
      ;FOLD ;%{H}
         Case 107
      ;ENDFOLD
      ;FOLD t9 ( EIN ) = STOP ;%{SE}%MKUKATPVW %CVW_SPS %VTSTOP %P 2:t9 ( EIN ) = STOP, 3: TSTOP
         VW(#SET_TIME,TRUE,9,1,0)
      ;ENDFOLD
      ;FOLD -- EZ3/SP3/KE3 oeffnen -- ;%{SE}%MKUKATPVW %CVW_COM %VCOMMENT %P 2:-- EZ3/SP3/KE3 oeffnen --, 3: VW_COMMENT
      ;ENDFOLD
      ;FOLD A1038 = AUS ;%{SE}%MKUKATPVW %CVW_SPS %VBOASG %P 2:A1038 = AUS, 3: BOASG
         $OUT[1038] = FALSE
      ;ENDFOLD
      ;FOLD A1086 = AUS ;%{SE}%MKUKATPVW %CVW_SPS %VBOASG %P 2:A1086 = AUS, 3: BOASG
         $OUT[1086] = FALSE
      ;ENDFOLD
      ;FOLD A1037 = EIN ;%{SE}%MKUKATPVW %CVW_SPS %VBOASG %P 2:A1037 = EIN, 3: BOASG
         $OUT[1037] = TRUE
      ;ENDFOLD
      ;FOLD -- KF3 Ausblasen -- ;%{SE}%MKUKATPVW %CVW_COM %VCOMMENT %P 2:-- KF3 Ausblasen --, 3: VW_COMMENT
      ;ENDFOLD
      ;FOLD A1156 = F330 + F331 + F332 + !F330 & !F331 & !F332 ;%{SE}%MKUKATPVW %CVW_SPS %VBOASG %P 2:A1156 = F330 + F331 + F332 + !F330 & !F331 & !F332, 3: BOASG
         $OUT[1156] = $FLAG[330] OR $FLAG[331] OR $FLAG[332] OR NOT $FLAG[330] AND NOT $FLAG[331] AND NOT $FLAG[332]
      ;ENDFOLD
      ;FOLD -- KF Ausblasen Ausschaltverzoegerung starten -- ;%{SE}%MKUKATPVW %CVW_COM %VCOMMENT %P 2:-- KF Ausblasen Ausschaltverzoegerung starten --, 3: VW_COMMENT
      ;ENDFOLD
      ;FOLD F739 = EIN ;%{SE}%MKUKATPVW %CVW_SPS %VBOASG %P 2:F739 = EIN, 3: BOASG
         $FLAG[739] = TRUE
      ;ENDFOLD
      ;FOLD -- RSK Sammelstoerung -- ;%{SE}%MKUKATPVW %CVW_COM %VCOMMENT %P 2:-- RSK Sammelstoerung --, 3: VW_COMMENT
      ;ENDFOLD
      ;FOLD F329 = T7 + T9 + F325 ;%{SE}%MKUKATPVW %CVW_SPS %VBOASG %P 2:F329 = T7 + T9 + F325, 3: BOASG
         $FLAG[329] = $TIMER_FLAG[7] OR $TIMER_FLAG[9] OR $FLAG[325]
      ;ENDFOLD
      ;FOLD -- Hilfsflag Startfraesen -- ;%{SE}%MKUKATPVW %CVW_COM %VCOMMENT %P 2:-- Hilfsflag Startfraesen --, 3: VW_COMMENT
      ;ENDFOLD
      ;FOLD F188 = (F188 & F174 + F190 & F175) & F287 ;%{SE}%MKUKATPVW %CVW_SPS %VBOASG %P 2:F188 = (F188 & F174 + F190 & F175) & F287, 3: BOASG
         $FLAG[188] = ($FLAG[188] AND $FLAG[174] OR $FLAG[190] AND $FLAG[175]) AND $FLAG[287]
      ;ENDFOLD
      ;FOLD F190 = !F200 & F190 + F200 & F287 & F190 ;%{SE}%MKUKATPVW %CVW_SPS %VBOASG %P 2:F190 = !F200 & F190 + F200 & F287 & F190, 3: BOASG
         $FLAG[190] = NOT $FLAG[200] AND $FLAG[190] OR $FLAG[200] AND $FLAG[287] AND $FLAG[190]
      ;ENDFOLD
      ;FOLD F287 = F174 + F175 & F200 ;%{SE}%MKUKATPVW %CVW_SPS %VBOASG %P 2:F287 = F174 + F175 & F200, 3: BOASG
         $FLAG[287] = $FLAG[174] OR $FLAG[175] AND $FLAG[200]
      ;ENDFOLD
      ;FOLD -- Neues Fraesprogramm und Zaehler ruecksetzen -- ;%{SE}%MKUKATPVW %CVW_COM %VCOMMENT %P 2:-- Neues Fraesprogramm und Zaehler ruecksetzen --, 3: VW_COMMENT
      ;ENDFOLD
      ;FOLD bin3 ( F200 ) = 36 ;%{SE}%MKUKATPVW %CVW_SPS %VARIASG %P 2:bin3 ( F200 ) = 36, 3: ARIASG
         VW(#BINOUT,$FLAG[200],3,36)
      ;ENDFOLD
      ;FOLD i19 ( F188 ) = i45 ;%{SE}%MKUKATPVW %CVW_SPS %VARIASG %P 2:i19 ( F188 ) = i45, 3: ARIASG
         VW(#COUNTER,$FLAG[188],19,$COUNT_I[45])
      ;ENDFOLD
      ;FOLD -- Wiederholung beim Startfraesen -- ;%{SE}%MKUKATPVW %CVW_COM %VCOMMENT %P 2:-- Wiederholung beim Startfraesen --, 3: VW_COMMENT
      ;ENDFOLD
      ;FOLD Schritt 104 = E1037 & !E1038 & (F174 & !F188 + F175 & F200 & !F188) & !F325 & !F329 & A4039 ;%{SE}%MKUKATPVW %CVW_SPS %VST_CON %P 2:Schritt 104 = E1037 & !E1038 & (F174 & !F188 + F175 & F200 & !F188) & !F325 & !F329 & A4039, 3: ST_CON
         IF $IN[1037] AND NOT $IN[1038] AND ($FLAG[174] AND NOT $FLAG[188] OR $FLAG[175] AND $FLAG[200] AND NOT $FLAG[188]) AND NOT $FLAG[325] AND NOT $FLAG[329] AND $OUT[4039] THEN
            PREVSTEP = $APP_INT[5]
            $APP_INT[5] = 104
         ENDIF
      ;ENDFOLD
      ;FOLD -- Weiter wenn Fraesen fertig -- ;%{SE}%MKUKATPVW %CVW_COM %VCOMMENT %P 2:-- Weiter wenn Fraesen fertig --, 3: VW_COMMENT
      ;ENDFOLD
      ;FOLD Schritt 108 = E1037 & !E1038 & (F175 & F190 & (!F200 + F188)+ F174 & F188 + F325 + F329) & A4039 ;%{SE}%MKUKATPVW %CVW_SPS %VST_CON %P 2:Schritt 108 = E1037 & !E1038 & (F175 & F190 & (!F200 + F188)+ F174 & F188 + F325 + F329) & A4039, 3: ST_CON
         IF $IN[1037] AND NOT $IN[1038] AND ($FLAG[175] AND $FLAG[190] AND (NOT $FLAG[200] OR $FLAG[188]) OR $FLAG[174] AND $FLAG[188] OR $FLAG[325] OR $FLAG[329]) AND $OUT[4039] THEN
            PREVSTEP = $APP_INT[5]
            $APP_INT[5] = 108
         ENDIF
      ;ENDFOLD
   ;ENDFOLD
   ;FOLD SCHRITT 108 -- STAT EZ3/SP3/KE3 -- ;%{P}%MKUKATPVW,%CSTEP,%VST_NR,%P 1:SCHRITT, 2:108, 3: STAT EZ3/SP3/KE3
      ;FOLD ;%{H}
         Case 108
      ;ENDFOLD
      ;FOLD F324 = AUS ;%{SE}%MKUKATPVW %CVW_SPS %VBOASG %P 2:F324 = AUS, 3: BOASG
         $FLAG[324] = FALSE
      ;ENDFOLD
      ;FOLD A1037 = AUS ;%{SE}%MKUKATPVW %CVW_SPS %VBOASG %P 2:A1037 = AUS, 3: BOASG
         $OUT[1037] = FALSE
      ;ENDFOLD
      ;FOLD -- KF3 abschalten -- ;%{SE}%MKUKATPVW %CVW_COM %VCOMMENT %P 2:-- KF3 abschalten --, 3: VW_COMMENT
      ;ENDFOLD
      ;FOLD A1154 = AUS ;%{SE}%MKUKATPVW %CVW_SPS %VBOASG %P 2:A1154 = AUS, 3: BOASG
         $OUT[1154] = FALSE
      ;ENDFOLD
      ;FOLD -- Ueberwachungszeit KF1 Versetzeinheit -- ;%{SE}%MKUKATPVW %CVW_COM %VCOMMENT %P 2:-- Ueberwachungszeit KF1 Versetzeinheit --, 3: VW_COMMENT
      ;ENDFOLD
      ;FOLD t8 ( EIN ) = -20[1/10Sek] ;%{SE}%MKUKATPVW %CVW_SPS %VTASG %P 2:t8 ( EIN ) = -20[1/10Sek], 3: TASG
         VW(#SET_TIME,TRUE,8,0,-20)
      ;ENDFOLD
      ;FOLD Schritt 109 = A4039 ;%{SE}%MKUKATPVW %CVW_SPS %VST_CON %P 2:Schritt 109 = A4039, 3: ST_CON
         IF $OUT[4039] THEN
            PREVSTEP = $APP_INT[5]
            $APP_INT[5] = 109
         ENDIF
      ;ENDFOLD
   ;ENDFOLD
   ;FOLD SCHRITT 109 -- STAT EZ3/SP3/KE3 -- ;%{P}%MKUKATPVW,%CSTEP,%VST_NR,%P 1:SCHRITT, 2:109, 3: STAT EZ3/SP3/KE3
      ;FOLD ;%{H}
         Case 109
      ;ENDFOLD
      ;FOLD F328 = AUS ;%{SE}%MKUKATPVW %CVW_SPS %VBOASG %P 2:F328 = AUS, 3: BOASG
         $FLAG[328] = FALSE
      ;ENDFOLD
      ;FOLD -- KF3 Versetzeinheit vor -- ;%{SE}%MKUKATPVW %CVW_COM %VCOMMENT %P 2:-- KF3 Versetzeinheit vor --, 3: VW_COMMENT
      ;ENDFOLD
      ;FOLD A1155 = F566 ;%{SE}%MKUKATPVW %CVW_SPS %VBOASG %P 2:A1155 = F566, 3: BOASG
         $OUT[1155] = $FLAG[566]
      ;ENDFOLD
      ;FOLD -- RSK Fehlerausgabe KS3 Arbeitsst. -- ;%{SE}%MKUKATPVW %CVW_COM %VCOMMENT %P 2:-- RSK Fehlerausgabe KS3 Arbeitsst. --, 3: VW_COMMENT
      ;ENDFOLD
      ;FOLD F324 = (E1156 + !E1157 + !E1158 + E1159) & !F323 & !F328 + F324 ;%{SE}%MKUKATPVW %CVW_SPS %VBOASG %P 2:F324 = (E1156 + !E1157 + !E1158 + E1159) & !F323 & !F328 + F324, 3: BOASG
         $FLAG[324] = ($IN[1156] OR NOT $IN[1157] OR NOT $IN[1158] OR $IN[1159]) AND NOT $FLAG[323] AND NOT $FLAG[328] OR $FLAG[324]
      ;ENDFOLD
      ;FOLD -- RSK Sammelstoerung -- ;%{SE}%MKUKATPVW %CVW_COM %VCOMMENT %P 2:-- RSK Sammelstoerung --, 3: VW_COMMENT
      ;ENDFOLD
      ;FOLD F329 = F324 + F325 ;%{SE}%MKUKATPVW %CVW_SPS %VBOASG %P 2:F329 = F324 + F325, 3: BOASG
         $FLAG[329] = $FLAG[324] OR $FLAG[325]
      ;ENDFOLD
      ;FOLD -- Ueberwachungszeit KS3 schwenken -- ;%{SE}%MKUKATPVW %CVW_COM %VCOMMENT %P 2:-- Ueberwachungszeit KS3 schwenken --, 3: VW_COMMENT
      ;ENDFOLD
      ;FOLD t9 ( EIN ) = -100[1/10Sek] ;%{SE}%MKUKATPVW %CVW_SPS %VTASG %P 2:t9 ( EIN ) = -100[1/10Sek], 3: TASG
         VW(#SET_TIME,TRUE,9,0,-100)
      ;ENDFOLD
      ;FOLD Schritt 108 = F324 & (E26 + E27) & A4039 ;%{SE}%MKUKATPVW %CVW_SPS %VST_CON %P 2:Schritt 108 = F324 & (E26 + E27) & A4039, 3: ST_CON
         IF $FLAG[324] AND ($IN[26] OR $IN[27]) AND $OUT[4039] THEN
            PREVSTEP = $APP_INT[5]
            $APP_INT[5] = 108
         ENDIF
      ;ENDFOLD
      ;FOLD Schritt 110 = (!F324 & (E1155 & F566 + !E1155 & !F566) + T8 + F325) & A4039 ;%{SE}%MKUKATPVW %CVW_SPS %VST_CON %P 2:Schritt 110 = (!F324 & (E1155 & F566 + !E1155 & !F566) + T8 + F325) & A4039, 3: ST_CON
         IF (NOT $FLAG[324] AND ($IN[1155] AND $FLAG[566] OR NOT $IN[1155] AND NOT $FLAG[566]) OR $TIMER_FLAG[8] OR $FLAG[325]) AND $OUT[4039] THEN
            PREVSTEP = $APP_INT[5]
            $APP_INT[5] = 110
         ENDIF
      ;ENDFOLD
   ;ENDFOLD
   ;FOLD SCHRITT 110 -- STAT EZ3/SP3/KE3-- ;%{P}%MKUKATPVW,%CSTEP,%VST_NR,%P 1:SCHRITT, 2:110, 3: STAT EZ3/SP3/KE3
      ;FOLD ;%{H}
         Case 110
      ;ENDFOLD
      ;FOLD F323 = AUS ;%{SE}%MKUKATPVW %CVW_SPS %VBOASG %P 2:F323 = AUS, 3: BOASG
         $FLAG[323] = FALSE
      ;ENDFOLD
      ;FOLD F328 = AUS ;%{SE}%MKUKATPVW %CVW_SPS %VBOASG %P 2:F328 = AUS, 3: BOASG
         $FLAG[328] = FALSE
      ;ENDFOLD
      ;FOLD -- RSK Sammelstoerung -- ;%{SE}%MKUKATPVW %CVW_COM %VCOMMENT %P 2:-- RSK Sammelstoerung --, 3: VW_COMMENT
      ;ENDFOLD
      ;FOLD F329 = F325 ;%{SE}%MKUKATPVW %CVW_SPS %VBOASG %P 2:F329 = F325, 3: BOASG
         $FLAG[329] = $FLAG[325]
      ;ENDFOLD
      ;FOLD -- KF3 ein -- ;%{SE}%MKUKATPVW %CVW_COM %VCOMMENT %P 2:-- KF3 ein --, 3: VW_COMMENT
      ;ENDFOLD
      ;FOLD A1154 = EIN ;%{SE}%MKUKATPVW %CVW_SPS %VBOASG %P 2:A1154 = EIN, 3: BOASG
         $OUT[1154] = TRUE
      ;ENDFOLD
      ;FOLD -- KS3 in Ruhestellung schwenken -- ;%{SE}%MKUKATPVW %CVW_COM %VCOMMENT %P 2:-- KS3 in Ruhestellung schwenken --, 3: VW_COMMENT
      ;ENDFOLD
      ;FOLD A1160 = (F747 + !F714) & E1037 & (E1155 & F566 + !E1155 & !F566) ;%{SE}%MKUKATPVW %CVW_SPS %VBOASG %P 2:A1160 = (F747 + !F714) & E1037 & (E1155 & F566 + !E1155 & !F566), 3: BOASG
         $OUT[1160] = ($FLAG[747] OR NOT $FLAG[714]) AND $IN[1037] AND ($IN[1155] AND $FLAG[566] OR NOT $IN[1155] AND NOT $FLAG[566])
      ;ENDFOLD
      ;FOLD Schritt 111 = (F747 + !F714 + T9) & (A1160 + T9) & E1037 & A4039 ;%{SE}%MKUKATPVW %CVW_SPS %VST_CON %P 2:Schritt 111 = (F747 + !F714 + T9) & (A1160 + T9) & E1037 & A4039, 3: ST_CON
         IF ($FLAG[747] OR NOT $FLAG[714] OR $TIMER_FLAG[9]) AND ($OUT[1160] OR $TIMER_FLAG[9]) AND $IN[1037] AND $OUT[4039] THEN
            PREVSTEP = $APP_INT[5]
            $APP_INT[5] = 111
         ENDIF
      ;ENDFOLD
   ;ENDFOLD
   ;FOLD SCHRITT 111 -- STAT EZ3/SP3/KE3 -- ;%{P}%MKUKATPVW,%CSTEP,%VST_NR,%P 1:SCHRITT, 2:111, 3: STAT EZ3/SP3/KE3
      ;FOLD ;%{H}
         Case 111
      ;ENDFOLD
      ;FOLD -- Hilfsflag SK Programmwechsel -- ;%{SE}%MKUKATPVW %CVW_COM %VCOMMENT %P 2:-- Hilfsflag SK Programmwechsel --, 3: VW_COMMENT
      ;ENDFOLD
      ;FOLD F334 = AUS ;%{SE}%MKUKATPVW %CVW_SPS %VBOASG %P 2:F334 = AUS, 3: BOASG
         $FLAG[334] = FALSE
      ;ENDFOLD
      ;FOLD -- RSK Fehlerausgabe KF Versetzeinheit -- ;%{SE}%MKUKATPVW %CVW_COM %VCOMMENT %P 2:-- RSK Fehlerausgabe KF Versetzeinheit --, 3: VW_COMMENT
      ;ENDFOLD
      ;FOLD F328 = !E1155 & F566 & !F323 + F328 ;%{SE}%MKUKATPVW %CVW_SPS %VBOASG %P 2:F328 = !E1155 & F566 & !F323 + F328, 3: BOASG
         $FLAG[328] = NOT $IN[1155] AND $FLAG[566] AND NOT $FLAG[323] OR $FLAG[328]
      ;ENDFOLD
      ;FOLD -- RSK Fehlerausgabe KS3 Ruhestellung -- ;%{SE}%MKUKATPVW %CVW_COM %VCOMMENT %P 2:-- RSK Fehlerausgabe KS3 Ruhestellung --, 3: VW_COMMENT
      ;ENDFOLD
      ;FOLD F323 = (!E1156 + E1157 + E1158 + !E1159) & T9 & (E1155 + !F566) + F323 ;%{SE}%MKUKATPVW %CVW_SPS %VBOASG %P 2:F323 = (!E1156 + E1157 + E1158 + !E1159) & T9 & (E1155 + !F566) + F323, 3: BOASG
         $FLAG[323] = (NOT $IN[1156] OR $IN[1157] OR $IN[1158] OR NOT $IN[1159]) AND $TIMER_FLAG[9] AND ($IN[1155] OR NOT $FLAG[566]) OR $FLAG[323]
      ;ENDFOLD
      ;FOLD -- RSK Fehlerausgabe EZ/SP min. Oeffnung -- ;%{SE}%MKUKATPVW %CVW_COM %VCOMMENT %P 2:-- RSK Fehlerausgabe EZ/SP min. Oeffnung --, 3: VW_COMMENT
      ;ENDFOLD
      ;FOLD F333 = !F747 ;%{SE}%MKUKATPVW %CVW_SPS %VBOASG %P 2:F333 = !F747, 3: BOASG
         $FLAG[333] = NOT $FLAG[747]
      ;ENDFOLD
      ;FOLD -- RSK Sammelstoerung -- ;%{SE}%MKUKATPVW %CVW_COM %VCOMMENT %P 2:-- RSK Sammelstoerung --, 3: VW_COMMENT
      ;ENDFOLD
      ;FOLD F329 = F323 + F325 + F328 ;%{SE}%MKUKATPVW %CVW_SPS %VBOASG %P 2:F329 = F323 + F325 + F328, 3: BOASG
         $FLAG[329] = $FLAG[323] OR $FLAG[325] OR $FLAG[328]
      ;ENDFOLD
      ;FOLD A1154 = !F323 & !F328 ;%{SE}%MKUKATPVW %CVW_SPS %VBOASG %P 2:A1154 = !F323 & !F328, 3: BOASG
         $OUT[1154] = NOT $FLAG[323] AND NOT $FLAG[328]
      ;ENDFOLD
      ;FOLD A1155 = F566 ;%{SE}%MKUKATPVW %CVW_SPS %VBOASG %P 2:A1155 = F566, 3: BOASG
         $OUT[1155] = $FLAG[566]
      ;ENDFOLD
      ;FOLD Schritt 109 = (F323 + F328) & (E26 + E27) & A4039 ;%{SE}%MKUKATPVW %CVW_SPS %VST_CON %P 2:Schritt 109 = (F323 + F328) & (E26 + E27) & A4039, 3: ST_CON
         IF ($FLAG[323] OR $FLAG[328]) AND ($IN[26] OR $IN[27]) AND $OUT[4039] THEN
            PREVSTEP = $APP_INT[5]
            $APP_INT[5] = 109
         ENDIF
      ;ENDFOLD
      ;FOLD Schritt 112 = !A1160 & E1156 & !E1157 & !E1158 & E1159 & A4039 ;%{SE}%MKUKATPVW %CVW_SPS %VST_CON %P 2:Schritt 112 = !A1160 & E1156 & !E1157 & !E1158 & E1159 & A4039, 3: ST_CON
         IF NOT $OUT[1160] AND $IN[1156] AND NOT $IN[1157] AND NOT $IN[1158] AND $IN[1159] AND $OUT[4039] THEN
            PREVSTEP = $APP_INT[5]
            $APP_INT[5] = 112
         ENDIF
      ;ENDFOLD
   ;ENDFOLD
   ;FOLD SCHRITT 112 -- STAT EZ3/SP3/KE3 -- ;%{P}%MKUKATPVW,%CSTEP,%VST_NR,%P 1:SCHRITT, 2:112, 3: STAT EZ3/SP3/KE3
      ;FOLD ;%{H}
         Case 112
      ;ENDFOLD
      ;FOLD F323 = AUS ;%{SE}%MKUKATPVW %CVW_SPS %VBOASG %P 2:F323 = AUS, 3: BOASG
         $FLAG[323] = FALSE
      ;ENDFOLD
      ;FOLD F328 = AUS ;%{SE}%MKUKATPVW %CVW_SPS %VBOASG %P 2:F328 = AUS, 3: BOASG
         $FLAG[328] = FALSE
      ;ENDFOLD
      ;FOLD -- RSK Sammelstoerung -- ;%{SE}%MKUKATPVW %CVW_COM %VCOMMENT %P 2:-- RSK Sammelstoerung --, 3: VW_COMMENT
      ;ENDFOLD
      ;FOLD F329 = F325 ;%{SE}%MKUKATPVW %CVW_SPS %VBOASG %P 2:F329 = F325, 3: BOASG
         $FLAG[329] = $FLAG[325]
      ;ENDFOLD
      ;FOLD t9 ( EIN ) = STOP ;%{SE}%MKUKATPVW %CVW_SPS %VTSTOP %P 2:t9 ( EIN ) = STOP, 3: TSTOP
         VW(#SET_TIME,TRUE,9,1,0)
      ;ENDFOLD
      ;FOLD -- KF1 Versetzeinheit rueck -- ;%{SE}%MKUKATPVW %CVW_COM %VCOMMENT %P 2:-- KF1 Versetzeinheit rueck --, 3: VW_COMMENT
      ;ENDFOLD
      ;FOLD A1155 = AUS ;%{SE}%MKUKATPVW %CVW_SPS %VBOASG %P 2:A1155 = AUS, 3: BOASG
         $OUT[1155] = FALSE
      ;ENDFOLD
      ;FOLD -- KF3 aus -- ;%{SE}%MKUKATPVW %CVW_COM %VCOMMENT %P 2:-- KF3 aus --, 3: VW_COMMENT
      ;ENDFOLD
      ;FOLD A1154 = AUS ;%{SE}%MKUKATPVW %CVW_SPS %VBOASG %P 2:A1154 = AUS, 3: BOASG
         $OUT[1154] = FALSE
      ;ENDFOLD
      ;FOLD -- KF1 Ausblasen -- ;%{SE}%MKUKATPVW %CVW_COM %VCOMMENT %P 2:-- KF1 Ausblasen --, 3: VW_COMMENT
      ;ENDFOLD
      ;FOLD A1166 = (F330 + F331 + F332) & F739 ;%{SE}%MKUKATPVW %CVW_SPS %VBOASG %P 2:A1166 = (F330 + F331 + F332) & F739, 3: BOASG
         $OUT[1166] = ($FLAG[330] OR $FLAG[331] OR $FLAG[332]) AND $FLAG[739]
      ;ENDFOLD
      ;FOLD bin9 ( !F329 ) = 1 ;%{SE}%MKUKATPVW %CVW_SPS %VARIASG %P 2:bin9 ( !F329 ) = 1, 3: ARIASG
         VW(#BINOUT,NOT $FLAG[329],9,1)
      ;ENDFOLD
      ;FOLD -- Wartezeit Programmwechsel SK -- ;%{SE}%MKUKATPVW %CVW_COM %VCOMMENT %P 2:-- Wartezeit Programmwechsel SK --, 3: VW_COMMENT
      ;ENDFOLD
      ;FOLD t8 ( !F334 ) = -2 [1/10Sek] ;%{SE}%MKUKATPVW %CVW_SPS %VTASG %P 2:t8 ( !F334 ) = -2 [1/10Sek], 3: TASG
         VW(#SET_TIME,NOT $FLAG[334],8,0,-2)
      ;ENDFOLD
      ;FOLD -- Hilfsflag SK Programmwechsel -- ;%{SE}%MKUKATPVW %CVW_COM %VCOMMENT %P 2:-- Hilfsflag SK Programmwechsel --, 3: VW_COMMENT
      ;ENDFOLD
      ;FOLD F334 = EIN ;%{SE}%MKUKATPVW %CVW_SPS %VBOASG %P 2:F334 = EIN, 3: BOASG
         $FLAG[334] = TRUE
      ;ENDFOLD
      ;FOLD -- Ueberwachungszeit EZ3/SP3/KE3 Messen -- ;%{SE}%MKUKATPVW %CVW_COM %VCOMMENT %P 2:-- Ueberwachungszeit EZ3/SP3/KE3 Messen --, 3: VW_COMMENT
      ;ENDFOLD
      ;FOLD t9 ( EIN ) = -150[1/10Sek] ;%{SE}%MKUKATPVW %CVW_SPS %VTASG %P 2:t9 ( EIN ) = -150[1/10Sek], 3: TASG
         VW(#SET_TIME,TRUE,9,0,-150)
      ;ENDFOLD
      ;FOLD Schritt 97 = (F325 + F329) & (E26 + E27) & A4039 ;%{SE}%MKUKATPVW %CVW_SPS %VST_CON %P 2:Schritt 97 = (F325 + F329) & (E26 + E27) & A4039, 3: ST_CON
         IF ($FLAG[325] OR $FLAG[329]) AND ($IN[26] OR $IN[27]) AND $OUT[4039] THEN
            PREVSTEP = $APP_INT[5]
            $APP_INT[5] = 97
         ENDIF
      ;ENDFOLD
      ;FOLD Schritt 113 = T8 & !F325 & !F329 & A4039 ;%{SE}%MKUKATPVW %CVW_SPS %VST_CON %P 2:Schritt 113 = T8 & !F325 & !F329 & A4039, 3: ST_CON
         IF $TIMER_FLAG[8] AND NOT $FLAG[325] AND NOT $FLAG[329] AND $OUT[4039] THEN
            PREVSTEP = $APP_INT[5]
            $APP_INT[5] = 113
         ENDIF
      ;ENDFOLD
   ;ENDFOLD
   ;FOLD SCHRITT 113 -- STAT EZ3/SP3/KE3 -- ;%{P}%MKUKATPVW,%CSTEP,%VST_NR,%P 1:SCHRITT, 2:113, 3: STAT EZ3/SP3/KE3
      ;FOLD ;%{H}
         Case 113
      ;ENDFOLD
      ;FOLD -- Hilfsflag SK Programmwechsel -- ;%{SE}%MKUKATPVW %CVW_COM %VCOMMENT %P 2:-- Hilfsflag SK Programmwechsel --, 3: VW_COMMENT
      ;ENDFOLD
      ;FOLD F334 = AUS ;%{SE}%MKUKATPVW %CVW_SPS %VBOASG %P 2:F334 = AUS, 3: BOASG
         $FLAG[334] = FALSE
      ;ENDFOLD
      ;FOLD -- Quitt. Fraesen SK3 -- ;%{SE}%MKUKATPVW %CVW_COM %VCOMMENT %P 2:-- Quitt. Fraesen SK3 --, 3: VW_COMMENT
      ;ENDFOLD
      ;FOLD A1106 = !F329 & !F322 ;%{SE}%MKUKATPVW %CVW_SPS %VBOASG %P 2:A1106 = !F329 & !F322, 3: BOASG
         $OUT[1106] = NOT $FLAG[329] AND NOT $FLAG[322]
      ;ENDFOLD
      ;FOLD -- RSK Sammelstoerung -- ;%{SE}%MKUKATPVW %CVW_COM %VCOMMENT %P 2:-- RSK Sammelstoerung --, 3: VW_COMMENT
      ;ENDFOLD
      ;FOLD F329 = T9 ;%{SE}%MKUKATPVW %CVW_SPS %VBOASG %P 2:F329 = T9, 3: BOASG
         $FLAG[329] = $TIMER_FLAG[9]
      ;ENDFOLD
      ;FOLD -- Messen nach Fraesen -- ;%{SE}%MKUKATPVW %CVW_COM %VCOMMENT %P 2:-- Messen nach Fraesen --, 3: VW_COMMENT
      ;ENDFOLD
      ;FOLD A1079 = !F174 & F175 ;%{SE}%MKUKATPVW %CVW_SPS %VBOASG %P 2:A1079 = !F174 & F175, 3: BOASG
         $OUT[1079] = NOT $FLAG[174] AND $FLAG[175]
      ;ENDFOLD
      ;FOLD A1078 = F174 & !F175 ;%{SE}%MKUKATPVW %CVW_SPS %VBOASG %P 2:A1078 = F174 & !F175, 3: BOASG
         $OUT[1078] = $FLAG[174] AND NOT $FLAG[175]
      ;ENDFOLD
      ;FOLD A1077 = (F174 + F175) & !F329 ;%{SE}%MKUKATPVW %CVW_SPS %VBOASG %P 2:A1077 = (F174 + F175) & !F329, 3: BOASG
         $OUT[1077] = ($FLAG[174] OR $FLAG[175]) AND NOT $FLAG[329]
      ;ENDFOLD
      ;FOLD Schritt 114 = !E1106 & E1107 & !E1108 & A4039 ;%{SE}%MKUKATPVW %CVW_SPS %VST_CON %P 2:Schritt 114 = !E1106 & E1107 & !E1108 & A4039, 3: ST_CON
         IF NOT $IN[1106] AND $IN[1107] AND NOT $IN[1108] AND $OUT[4039] THEN
            PREVSTEP = $APP_INT[5]
            $APP_INT[5] = 114
         ENDIF
      ;ENDFOLD
   ;ENDFOLD
   ;FOLD SCHRITT 114 -- STAT EZ3/SP3/KE3 -- ;%{P}%MKUKATPVW,%CSTEP,%VST_NR,%P 1:SCHRITT, 2:114, 3: STAT EZ3/SP3/KE3
      ;FOLD ;%{H}
         Case 114
      ;ENDFOLD
      ;FOLD -- Hilfsflag SK Programmwechsel -- ;%{SE}%MKUKATPVW %CVW_COM %VCOMMENT %P 2:-- Hilfsflag SK Programmwechsel --, 3: VW_COMMENT
      ;ENDFOLD
      ;FOLD F334 = AUS ;%{SE}%MKUKATPVW %CVW_SPS %VBOASG %P 2:F334 = AUS, 3: BOASG
         $FLAG[334] = FALSE
      ;ENDFOLD
      ;FOLD -- RSK Sammelstoerung -- ;%{SE}%MKUKATPVW %CVW_COM %VCOMMENT %P 2:-- RSK Sammelstoerung --, 3: VW_COMMENT
      ;ENDFOLD
      ;FOLD F329 = T9 ;%{SE}%MKUKATPVW %CVW_SPS %VBOASG %P 2:F329 = T9, 3: BOASG
         $FLAG[329] = $TIMER_FLAG[9]
      ;ENDFOLD
      ;FOLD Schritt 115 = E1037 & (E1077 & !E1096 + T9) & A4039 ;%{SE}%MKUKATPVW %CVW_SPS %VST_CON %P 2:Schritt 115 = E1037 & (E1077 & !E1096 + T9) & A4039, 3: ST_CON
         IF $IN[1037] AND ($IN[1077] AND NOT $IN[1096] OR $TIMER_FLAG[9]) AND $OUT[4039] THEN
            PREVSTEP = $APP_INT[5]
            $APP_INT[5] = 115
         ENDIF
      ;ENDFOLD
   ;ENDFOLD
   ;FOLD SCHRITT 115 -- STAT EZ3/SP3/KE3 -- ;%{P}%MKUKATPVW,%CSTEP,%VST_NR,%P 1:SCHRITT, 2:115, 3: STAT EZ3/SP3/KE3
      ;FOLD ;%{H}
         Case 115
      ;ENDFOLD
      ;FOLD t9 ( EIN ) = STOP ;%{SE}%MKUKATPVW %CVW_SPS %VTSTOP %P 2:t9 ( EIN ) = STOP, 3: TSTOP
         VW(#SET_TIME,TRUE,9,1,0)
      ;ENDFOLD
      ;FOLD -- RSK Fehlerausgabe Kappenverschleiss -- ;%{SE}%MKUKATPVW %CVW_COM %VCOMMENT %P 2:-- RSK Fehlerausgabe Kappenverschleiss --, 3: VW_COMMENT
      ;ENDFOLD
      ;FOLD F196 = E1097 ;%{SE}%MKUKATPVW %CVW_SPS %VBOASG %P 2:F196 = E1097, 3: BOASG
         $FLAG[196] = $IN[1097]
      ;ENDFOLD
      ;FOLD -- RSK Fehlerausgabe Messen -- ;%{SE}%MKUKATPVW %CVW_COM %VCOMMENT %P 2:-- RSK Fehlerausgabe Messen --, 3: VW_COMMENT
      ;ENDFOLD
      ;FOLD F326 = E1096 + E1097 + E1098 + F326 ;%{SE}%MKUKATPVW %CVW_SPS %VBOASG %P 2:F326 = E1096 + E1097 + E1098 + F326, 3: BOASG
         $FLAG[326] = $IN[1096] OR $IN[1097] OR $IN[1098] OR $FLAG[326]
      ;ENDFOLD
      ;FOLD -- RSK Sammelstoerung -- ;%{SE}%MKUKATPVW %CVW_COM %VCOMMENT %P 2:-- RSK Sammelstoerung --, 3: VW_COMMENT
      ;ENDFOLD
      ;FOLD F329 = F326 ;%{SE}%MKUKATPVW %CVW_SPS %VBOASG %P 2:F329 = F326, 3: BOASG
         $FLAG[329] = $FLAG[326]
      ;ENDFOLD
      ;FOLD A1078 = AUS ;%{SE}%MKUKATPVW %CVW_SPS %VBOASG %P 2:A1078 = AUS, 3: BOASG
         $OUT[1078] = FALSE
      ;ENDFOLD
      ;FOLD A1079 = AUS ;%{SE}%MKUKATPVW %CVW_SPS %VBOASG %P 2:A1079 = AUS, 3: BOASG
         $OUT[1079] = FALSE
      ;ENDFOLD
      ;FOLD -- Druckvorgabe SK3/EZ3/SP3/KE3 -- ;%{SE}%MKUKATPVW %CVW_COM %VCOMMENT %P 2:-- Druckvorgabe SK3/EZ3/SP3/KE3 --, 3: VW_COMMENT
      ;ENDFOLD
      ;FOLD F168 = F174 & !F832 ;%{SE}%MKUKATPVW %CVW_SPS %VBOASG %P 2:F168 = F174 & !F832, 3: BOASG
         $FLAG[168] = $FLAG[174] AND NOT $FLAG[832]
      ;ENDFOLD
      ;FOLD bin7 ( F168 ) = 41 ;%{SE}%MKUKATPVW %CVW_SPS %VARIASG %P 2:bin7 ( F168 ) = 41, 3: ARIASG
         VW(#BINOUT,$FLAG[168],7,41)
      ;ENDFOLD
      ;FOLD F168 = F175 & !F832 ;%{SE}%MKUKATPVW %CVW_SPS %VBOASG %P 2:F168 = F175 & !F832, 3: BOASG
         $FLAG[168] = $FLAG[175] AND NOT $FLAG[832]
      ;ENDFOLD
      ;FOLD bin7 ( F168 ) = 51 ;%{SE}%MKUKATPVW %CVW_SPS %VARIASG %P 2:bin7 ( F168 ) = 51, 3: ARIASG
         VW(#BINOUT,$FLAG[168],7,51)
      ;ENDFOLD
      ;FOLD F168 = AUS ;%{SE}%MKUKATPVW %CVW_SPS %VBOASG %P 2:F168 = AUS, 3: BOASG
         $FLAG[168] = FALSE
      ;ENDFOLD
      ;FOLD bin9 ( F174 ) = 41 ;%{SE}%MKUKATPVW %CVW_SPS %VARIASG %P 2:bin9 ( F174 ) = 41, 3: ARIASG
         VW(#BINOUT,$FLAG[174],9,41)
      ;ENDFOLD
      ;FOLD bin9 ( F175 ) = 51 ;%{SE}%MKUKATPVW %CVW_SPS %VARIASG %P 2:bin9 ( F175 ) = 51, 3: ARIASG
         VW(#BINOUT,$FLAG[175],9,51)
      ;ENDFOLD
      ;FOLD -- Wartezeit Programmwechsel SK -- ;%{SE}%MKUKATPVW %CVW_COM %VCOMMENT %P 2:-- Wartezeit Programmwechsel SK --, 3: VW_COMMENT
      ;ENDFOLD
      ;FOLD T8 ( !F334 ) = -2[1/10Sek] ;%{SE}%MKUKATPVW %CVW_SPS %VTASG %P 2:T8 ( !F334 ) = -2[1/10Sek], 3: TASG
         VW(#SET_TIME,NOT $FLAG[334],8,0,-2)
      ;ENDFOLD
      ;FOLD -- Hilfsflag SK Programmwechsel -- ;%{SE}%MKUKATPVW %CVW_COM %VCOMMENT %P 2:-- Hilfsflag SK Programmwechsel --, 3: VW_COMMENT
      ;ENDFOLD
      ;FOLD F334 = EIN ;%{SE}%MKUKATPVW %CVW_SPS %VBOASG %P 2:F334 = EIN, 3: BOASG
         $FLAG[334] = TRUE
      ;ENDFOLD
      ;FOLD -- Ueberwachungszeit EZ3/SP3/KE3 Setzhub 2 -- ;%{SE}%MKUKATPVW %CVW_COM %VCOMMENT %P 2:-- Ueberwachungszeit EZ3/SP3/KE3 Setzhub 2 --, 3: VW_COMMENT
      ;ENDFOLD
      ;FOLD t9 ( EIN ) = -80[1/10Sek] ;%{SE}%MKUKATPVW %CVW_SPS %VTASG %P 2:t9 ( EIN ) = -80[1/10Sek], 3: TASG
         VW(#SET_TIME,TRUE,9,0,-80)
      ;ENDFOLD
      ;FOLD Schritt 116 = T8 & !F335 & A4039 ;%{SE}%MKUKATPVW %CVW_SPS %VST_CON %P 2:Schritt 116 = T8 & !F335 & A4039, 3: ST_CON
         IF $TIMER_FLAG[8] AND NOT $FLAG[335] AND $OUT[4039] THEN
            PREVSTEP = $APP_INT[5]
            $APP_INT[5] = 116
         ENDIF
      ;ENDFOLD
      ;FOLD Schritt 116 = T8 & F335 & !F174 & A4039 ;%{SE}%MKUKATPVW %CVW_SPS %VST_CON %P 2:Schritt 116 = T8 & F335 & !F174 & A4039, 3: ST_CON
         IF $TIMER_FLAG[8] AND $FLAG[335] AND NOT $FLAG[174] AND $OUT[4039] THEN
            PREVSTEP = $APP_INT[5]
            $APP_INT[5] = 116
         ENDIF
      ;ENDFOLD
      ;FOLD Schritt 227 = T8 & F335 & F174 & A4039 ;%{SE}%MKUKATPVW %CVW_SPS %VST_CON %P 2:Schritt 227 = T8 & F335 & F174 & A4039, 3: ST_CON
         IF $TIMER_FLAG[8] AND $FLAG[335] AND $FLAG[174] AND $OUT[4039] THEN
            PREVSTEP = $APP_INT[5]
            $APP_INT[5] = 227
         ENDIF
      ;ENDFOLD
   ;ENDFOLD
   ;FOLD SCHRITT 116 -- STAT EZ3/SP3/KE3 -- ;%{P}%MKUKATPVW,%CSTEP,%VST_NR,%P 1:SCHRITT, 2:116, 3: STAT EZ3/SP3/KE3
      ;FOLD ;%{H}
         Case 116
      ;ENDFOLD
      ;FOLD -- Hilfsflag SK Programmwechsel -- ;%{SE}%MKUKATPVW %CVW_COM %VCOMMENT %P 2:-- Hilfsflag SK Programmwechsel --, 3: VW_COMMENT
      ;ENDFOLD
      ;FOLD F334 = AUS ;%{SE}%MKUKATPVW %CVW_SPS %VBOASG %P 2:F334 = AUS, 3: BOASG
         $FLAG[334] = FALSE
      ;ENDFOLD
      ;FOLD A1077 = AUS ;%{SE}%MKUKATPVW %CVW_SPS %VBOASG %P 2:A1077 = AUS, 3: BOASG
         $OUT[1077] = FALSE
      ;ENDFOLD
      ;FOLD -- EZ3/SP3/KE3 schliessen -- ;%{SE}%MKUKATPVW %CVW_COM %VCOMMENT %P 2:-- EZ3/SP3/KE3 schliessen --, 3: VW_COMMENT
      ;ENDFOLD
      ;FOLD A1037 = AUS ;%{SE}%MKUKATPVW %CVW_SPS %VBOASG %P 2:A1037 = AUS, 3: BOASG
         $OUT[1037] = FALSE
      ;ENDFOLD
      ;FOLD A1038 = !F329 & !F196 ;%{SE}%MKUKATPVW %CVW_SPS %VBOASG %P 2:A1038 = !F329 & !F196, 3: BOASG
         $OUT[1038] = NOT $FLAG[329] AND NOT $FLAG[196]
      ;ENDFOLD
      ;FOLD -- Ueberwachungszeit Kurzschlussschweissung SK3 -- ;%{SE}%MKUKATPVW %CVW_COM %VCOMMENT %P 2:-- Ueberwachungszeit Kurzschlussschweissung SK3 --, 3: VW_COMMENT
      ;ENDFOLD
      ;FOLD t9 ( EIN ) = -80[1/10Sek] ;%{SE}%MKUKATPVW %CVW_SPS %VTASG %P 2:t9 ( EIN ) = -80[1/10Sek], 3: TASG
         VW(#SET_TIME,TRUE,9,0,-80)
      ;ENDFOLD
      ;FOLD Schritt 117 = !E1037 & E1038 + E1037 & !E1038 & (F329 + F326 + F196) & A4039 ;%{SE}%MKUKATPVW %CVW_SPS %VST_CON %P 2:Schritt 117 = !E1037 & E1038 + E1037 & !E1038 & (F329 + F326 + F196) & A4039, 3: ST_CON
         IF NOT $IN[1037] AND $IN[1038] OR $IN[1037] AND NOT $IN[1038] AND ($FLAG[329] OR $FLAG[326] OR $FLAG[196]) AND $OUT[4039] THEN
            PREVSTEP = $APP_INT[5]
            $APP_INT[5] = 117
         ENDIF
      ;ENDFOLD
   ;ENDFOLD
   ;FOLD SCHRITT 117 -- STAT EZ3/SP3/KE3-- ;%{P}%MKUKATPVW,%CSTEP,%VST_NR,%P 1:SCHRITT, 2:117, 3: STAT EZ3/SP3/KE3
      ;FOLD ;%{H}
         Case 117
      ;ENDFOLD
      ;FOLD -- Hilfsflag SK Programmwechsel -- ;%{SE}%MKUKATPVW %CVW_COM %VCOMMENT %P 2:-- Hilfsflag SK Programmwechsel --, 3: VW_COMMENT
      ;ENDFOLD
      ;FOLD F334 = AUS ;%{SE}%MKUKATPVW %CVW_SPS %VBOASG %P 2:F334 = AUS, 3: BOASG
         $FLAG[334] = FALSE
      ;ENDFOLD
      ;FOLD t9 ( EIN ) = STOP ;%{SE}%MKUKATPVW %CVW_SPS %VTSTOP %P 2:t9 ( EIN ) = STOP, 3: TSTOP
         VW(#SET_TIME,TRUE,9,1,0)
      ;ENDFOLD
      ;FOLD -- RSK Fehlerausgabe Kraftaufbau -- ;%{SE}%MKUKATPVW %CVW_COM %VCOMMENT %P 2:-- RSK Fehlerausgabe Kraftaufbau --, 3: VW_COMMENT
      ;ENDFOLD
      ;FOLD F325 = T9 + F325 ;%{SE}%MKUKATPVW %CVW_SPS %VBOASG %P 2:F325 = T9 + F325, 3: BOASG
         $FLAG[325] = $TIMER_FLAG[9] OR $FLAG[325]
      ;ENDFOLD
      ;FOLD -- RSK Fehlerausgabe K -- ;%{SE}%MKUKATPVW %CVW_COM %VCOMMENT %P 2:-- RSK Fehlerausgabe K --, 3: VW_COMMENT
      ;ENDFOLD
      ;FOLD F327 = (A1105 & !F832 + A1038 & F831) & (E1125 + !E1122) + F327 ;%{SE}%MKUKATPVW %CVW_SPS %VBOASG %P 2:F327 = (A1105 & !F832 + A1038 & F831) & (E1125 + !E1122) + F327, 3: BOASG
         $FLAG[327] = ($OUT[1105] AND NOT $FLAG[832] OR $OUT[1038] AND $FLAG[831]) AND ($IN[1125] OR NOT $IN[1122]) OR $FLAG[327]
      ;ENDFOLD
      ;FOLD -- RSK Sammelstoerung -- ;%{SE}%MKUKATPVW %CVW_COM %VCOMMENT %P 2:-- RSK Sammelstoerung --, 3: VW_COMMENT
      ;ENDFOLD
      ;FOLD F329 = F325 + F326 + F327 ;%{SE}%MKUKATPVW %CVW_SPS %VBOASG %P 2:F329 = F325 + F326 + F327, 3: BOASG
         $FLAG[329] = $FLAG[325] OR $FLAG[326] OR $FLAG[327]
      ;ENDFOLD
      ;FOLD -- Kurzschlussschweissung SK3 -- ;%{SE}%MKUKATPVW %CVW_COM %VCOMMENT %P 2:-- Kurzschlussschweissung SK3 --, 3: VW_COMMENT
      ;ENDFOLD
      ;FOLD A1105 = !F325 & !F329 & !F196 ;%{SE}%MKUKATPVW %CVW_SPS %VBOASG %P 2:A1105 = !F325 & !F329 & !F196, 3: BOASG
         $OUT[1105] = NOT $FLAG[325] AND NOT $FLAG[329] AND NOT $FLAG[196]
      ;ENDFOLD
      ;FOLD -- Flagbildng Wiederholfraesen -- ;%{SE}%MKUKATPVW %CVW_COM %VCOMMENT %P 2:-- Flagbildng Wiederholfraesen --, 3: VW_COMMENT
      ;ENDFOLD
      ;FOLD F749 = (F322 + F323 + F325 + F326 + F327 + F329) & !F748 ;%{SE}%MKUKATPVW %CVW_SPS %VBOASG %P 2:F749 = (F322 + F323 + F325 + F326 + F327 + F329) & !F748, 3: BOASG
         $FLAG[749] = ($FLAG[322] OR $FLAG[323] OR $FLAG[325] OR $FLAG[326] OR $FLAG[327] OR $FLAG[329]) AND NOT $FLAG[748]
      ;ENDFOLD
      ;FOLD Schritt 97 = E1037 & !E1038 & (F322 + F323 + F325 + F326 + F327 + F329) & (E26 + E27) & A4039 ;%{SE}%MKUKATPVW %CVW_SPS %VST_CON %P 2:Schritt 97 = E1037 & !E1038 & (F322 + F323 + F325 + F326 + F327 + F329) & (E26 + E27) & A4039, 3: ST_CON
         IF $IN[1037] AND NOT $IN[1038] AND ($FLAG[322] OR $FLAG[323] OR $FLAG[325] OR $FLAG[326] OR $FLAG[327] OR $FLAG[329]) AND ($IN[26] OR $IN[27]) AND $OUT[4039] THEN
            PREVSTEP = $APP_INT[5]
            $APP_INT[5] = 97
         ENDIF
      ;ENDFOLD
      ;FOLD Schritt 118 = (E1105 & E1124 & !E1126 + E1105 & E15 + F326 + F327 + F196) & A4039 ;%{SE}%MKUKATPVW %CVW_SPS %VST_CON %P 2:Schritt 118 = (E1105 & E1124 & !E1126 + E1105 & E15 + F326 + F327 + F196) & A4039, 3: ST_CON
         IF ($IN[1105] AND $IN[1124] AND NOT $IN[1126] OR $IN[1105] AND $IN[15] OR $FLAG[326] OR $FLAG[327] OR $FLAG[196]) AND $OUT[4039] THEN
            PREVSTEP = $APP_INT[5]
            $APP_INT[5] = 118
         ENDIF
      ;ENDFOLD
   ;ENDFOLD
   ;FOLD SCHRITT 118 -- STAT EZ3/SP3/KE3 -- ;%{P}%MKUKATPVW,%CSTEP,%VST_NR,%P 1:SCHRITT, 2:118, 3: STAT EZ3/SP3/KE3
      ;FOLD ;%{H}
         Case 118
      ;ENDFOLD
      ;FOLD A1105 = AUS ;%{SE}%MKUKATPVW %CVW_SPS %VBOASG %P 2:A1105 = AUS, 3: BOASG
         $OUT[1105] = FALSE
      ;ENDFOLD
      ;FOLD F174 = !F327 & F174 ;%{SE}%MKUKATPVW %CVW_SPS %VBOASG %P 2:F174 = !F327 & F174, 3: BOASG
         $FLAG[174] = NOT $FLAG[327] AND $FLAG[174]
      ;ENDFOLD
      ;FOLD F175 = F327 + F175 ;%{SE}%MKUKATPVW %CVW_SPS %VBOASG %P 2:F175 = F327 + F175, 3: BOASG
         $FLAG[175] = $FLAG[327] OR $FLAG[175]
      ;ENDFOLD
      ;FOLD -- EZ3/SP3/KE3 oeffnen -- ;%{SE}%MKUKATPVW %CVW_COM %VCOMMENT %P 2:-- EZ3/SP3/KE3 oeffnen --, 3: VW_COMMENT
      ;ENDFOLD
      ;FOLD A1038 = AUS ;%{SE}%MKUKATPVW %CVW_SPS %VBOASG %P 2:A1038 = AUS, 3: BOASG
         $OUT[1038] = FALSE
      ;ENDFOLD
      ;FOLD A1037 = !E1037 ;%{SE}%MKUKATPVW %CVW_SPS %VBOASG %P 2:A1037 = !E1037, 3: BOASG
         $OUT[1037] = NOT $IN[1037]
      ;ENDFOLD
      ;FOLD bin9 ( !F326 ) = 1 ;%{SE}%MKUKATPVW %CVW_SPS %VARIASG %P 2:bin9 ( !F326 ) = 1, 3: ARIASG
         VW(#BINOUT,NOT $FLAG[326],9,1)
      ;ENDFOLD
      ;FOLD -- Wartezeit Programmwechsel SK -- ;%{SE}%MKUKATPVW %CVW_COM %VCOMMENT %P 2:-- Wartezeit Programmwechsel SK --, 3: VW_COMMENT
      ;ENDFOLD
      ;FOLD T8 ( !F334 ) = -2[1/10Sek] ;%{SE}%MKUKATPVW %CVW_SPS %VTASG %P 2:T8 ( !F334 ) = -2[1/10Sek], 3: TASG
         VW(#SET_TIME,NOT $FLAG[334],8,0,-2)
      ;ENDFOLD
      ;FOLD -- Hilfsflag SK Programmwechsel -- ;%{SE}%MKUKATPVW %CVW_COM %VCOMMENT %P 2:-- Hilfsflag SK Programmwechsel --, 3: VW_COMMENT
      ;ENDFOLD
      ;FOLD F334 = EIN ;%{SE}%MKUKATPVW %CVW_SPS %VBOASG %P 2:F334 = EIN, 3: BOASG
         $FLAG[334] = TRUE
      ;ENDFOLD
      ;FOLD F748 = F322 + F323 + F325 + F326 + F327 + F329 ;%{SE}%MKUKATPVW %CVW_SPS %VBOASG %P 2:F748 = F322 + F323 + F325 + F326 + F327 + F329, 3: BOASG
         $FLAG[748] = $FLAG[322] OR $FLAG[323] OR $FLAG[325] OR $FLAG[326] OR $FLAG[327] OR $FLAG[329]
      ;ENDFOLD
      ;FOLD Schritt 97 = E1037 & !E1038 & (F322 + F323 + F325 + F326 + F327 + F329) & (E26 + E27) & A4039 ;%{SE}%MKUKATPVW %CVW_SPS %VST_CON %P 2:Schritt 97 = E1037 & !E1038 & (F322 + F323 + F325 + F326 + F327 + F329) & (E26 + E27) & A4039, 3: ST_CON
         IF $IN[1037] AND NOT $IN[1038] AND ($FLAG[322] OR $FLAG[323] OR $FLAG[325] OR $FLAG[326] OR $FLAG[327] OR $FLAG[329]) AND ($IN[26] OR $IN[27]) AND $OUT[4039] THEN
            PREVSTEP = $APP_INT[5]
            $APP_INT[5] = 97
         ENDIF
      ;ENDFOLD
      ;FOLD Schritt 97 = E1037 & !E1038 & (F322 + F323 + F325 + F326 + F327 + F329) & (F731 & F749) & A4039 ;%{SE}%MKUKATPVW %CVW_SPS %VST_CON %P 2:Schritt 97 = E1037 & !E1038 & (F322 + F323 + F325 + F326 + F327 + F329) & (F731 & F749) & A4039, 3: ST_CON
         IF $IN[1037] AND NOT $IN[1038] AND ($FLAG[322] OR $FLAG[323] OR $FLAG[325] OR $FLAG[326] OR $FLAG[327] OR $FLAG[329]) AND ($FLAG[731] AND $FLAG[749]) AND $OUT[4039] THEN
            PREVSTEP = $APP_INT[5]
            $APP_INT[5] = 97
         ENDIF
      ;ENDFOLD
      ;FOLD Schritt 119 = T8 & E1037 & !E1038 & (!F325 & !F326 & !F327 & !F329 + F196) & A4039 ;%{SE}%MKUKATPVW %CVW_SPS %VST_CON %P 2:Schritt 119 = T8 & E1037 & !E1038 & (!F325 & !F326 & !F327 & !F329 + F196) & A4039, 3: ST_CON
         IF $TIMER_FLAG[8] AND $IN[1037] AND NOT $IN[1038] AND (NOT $FLAG[325] AND NOT $FLAG[326] AND NOT $FLAG[327] AND NOT $FLAG[329] OR $FLAG[196]) AND $OUT[4039] THEN
            PREVSTEP = $APP_INT[5]
            $APP_INT[5] = 119
         ENDIF
      ;ENDFOLD
   ;ENDFOLD
   ;FOLD SCHRITT 119 -- STAT EZ3/SP3/KE3 # Ende -- ;%{P}%MKUKATPVW,%CSTEP,%VST_NR,%P 1:SCHRITT, 2:119, 3: STAT EZ3/SP3/KE3 # Ende
      ;FOLD ;%{H}
         Case 119
      ;ENDFOLD
      ;FOLD -- Hilfsflag SK Programmwechsel -- ;%{SE}%MKUKATPVW %CVW_COM %VCOMMENT %P 2:-- Hilfsflag SK Programmwechsel --, 3: VW_COMMENT
      ;ENDFOLD
      ;FOLD F334 = AUS ;%{SE}%MKUKATPVW %CVW_SPS %VBOASG %P 2:F334 = AUS, 3: BOASG
         $FLAG[334] = FALSE
      ;ENDFOLD
      ;FOLD -- RSK Sammelstoerung -- ;%{SE}%MKUKATPVW %CVW_COM %VCOMMENT %P 2:-- RSK Sammelstoerung --, 3: VW_COMMENT
      ;ENDFOLD
      ;FOLD F329 = F196 ;%{SE}%MKUKATPVW %CVW_SPS %VBOASG %P 2:F329 = F196, 3: BOASG
         $FLAG[329] = $FLAG[196]
      ;ENDFOLD
      ;FOLD F185 = !E1106 & !E1108 + F196 & (E26 + E27) ;%{SE}%MKUKATPVW %CVW_SPS %VBOASG %P 2:F185 = !E1106 & !E1108 + F196 & (E26 + E27), 3: BOASG
         $FLAG[185] = NOT $IN[1106] AND NOT $IN[1108] OR $FLAG[196] AND ($IN[26] OR $IN[27])
      ;ENDFOLD
      ;FOLD Schritt 1 = F185 & A4039 ;%{SE}%MKUKATPVW %CVW_SPS %VST_CON %P 2:Schritt 1 = F185 & A4039, 3: ST_CON
         IF $FLAG[185] AND $OUT[4039] THEN
            PREVSTEP = $APP_INT[5]
            $APP_INT[5] = 1
         ENDIF
      ;ENDFOLD
   ;ENDFOLD
   ;FOLD SCHRITT 120 -- ROB STP1 SZ1 # Start -- ;%{P}%MKUKATPVW,%CSTEP,%VST_NR,%P 1:SCHRITT, 2:120, 3: ROB STP1 SZ1 # Start
      ;FOLD ;%{H}
         Case 120
      ;ENDFOLD
      ;FOLD -- RSK gestartet -- ;%{SE}%MKUKATPVW %CVW_COM %VCOMMENT %P 2:-- RSK gestartet --, 3: VW_COMMENT
      ;ENDFOLD
      ;FOLD F321 = AUS ;%{SE}%MKUKATPVW %CVW_SPS %VBOASG %P 2:F321 = AUS, 3: BOASG
         $FLAG[321] = FALSE
      ;ENDFOLD
      ;FOLD F122 = AUS ;%{SE}%MKUKATPVW %CVW_SPS %VBOASG %P 2:F122 = AUS, 3: BOASG
         $FLAG[122] = FALSE
      ;ENDFOLD
      ;FOLD F322 = AUS ;%{SE}%MKUKATPVW %CVW_SPS %VBOASG %P 2:F322 = AUS, 3: BOASG
         $FLAG[322] = FALSE
      ;ENDFOLD
      ;FOLD F323 = AUS ;%{SE}%MKUKATPVW %CVW_SPS %VBOASG %P 2:F323 = AUS, 3: BOASG
         $FLAG[323] = FALSE
      ;ENDFOLD
      ;FOLD F324 = AUS ;%{SE}%MKUKATPVW %CVW_SPS %VBOASG %P 2:F324 = AUS, 3: BOASG
         $FLAG[324] = FALSE
      ;ENDFOLD
      ;FOLD F325 = AUS ;%{SE}%MKUKATPVW %CVW_SPS %VBOASG %P 2:F325 = AUS, 3: BOASG
         $FLAG[325] = FALSE
      ;ENDFOLD
      ;FOLD F329 = AUS ;%{SE}%MKUKATPVW %CVW_SPS %VBOASG %P 2:F329 = AUS, 3: BOASG
         $FLAG[329] = FALSE
      ;ENDFOLD
      ;FOLD -- EZ1/SP1/KE1/STP1 SZ1 Zaehler -- ;%{SE}%MKUKATPVW %CVW_COM %VCOMMENT %P 2:-- EZ1/SP1/KE1/STP1 SZ1 Zaehler --, 3: VW_COMMENT
      ;ENDFOLD
      ;FOLD F94 = AUS ;%{SE}%MKUKATPVW %CVW_SPS %VBOASG %P 2:F94 = AUS, 3: BOASG
         $FLAG[94] = FALSE
      ;ENDFOLD
      ;FOLD F95 = AUS ;%{SE}%MKUKATPVW %CVW_SPS %VBOASG %P 2:F95 = AUS, 3: BOASG
         $FLAG[95] = FALSE
      ;ENDFOLD
      ;FOLD F96 = AUS ;%{SE}%MKUKATPVW %CVW_SPS %VBOASG %P 2:F96 = AUS, 3: BOASG
         $FLAG[96] = FALSE
      ;ENDFOLD
      ;FOLD F97 = AUS ;%{SE}%MKUKATPVW %CVW_SPS %VBOASG %P 2:F97 = AUS, 3: BOASG
         $FLAG[97] = FALSE
      ;ENDFOLD
      ;FOLD F98 = AUS ;%{SE}%MKUKATPVW %CVW_SPS %VBOASG %P 2:F98 = AUS, 3: BOASG
         $FLAG[98] = FALSE
      ;ENDFOLD
      ;FOLD F99 = AUS ;%{SE}%MKUKATPVW %CVW_SPS %VBOASG %P 2:F99 = AUS, 3: BOASG
         $FLAG[99] = FALSE
      ;ENDFOLD
      ;FOLD -- Hilfsflags Funktionstest KF Motor -- ;%{SE}%MKUKATPVW %CVW_COM %VCOMMENT %P 2:-- Hilfsflags Funktionstest KF Motor --, 3: VW_COMMENT
      ;ENDFOLD
      ;FOLD F312 = AUS ;%{SE}%MKUKATPVW %CVW_SPS %VBOASG %P 2:F312 = AUS, 3: BOASG
         $FLAG[312] = FALSE
      ;ENDFOLD
      ;FOLD F313 = AUS ;%{SE}%MKUKATPVW %CVW_SPS %VBOASG %P 2:F313 = AUS, 3: BOASG
         $FLAG[313] = FALSE
      ;ENDFOLD
      ;FOLD -- Ueberwachungszeit KF1 hochfahren -- ;%{SE}%MKUKATPVW %CVW_COM %VCOMMENT %P 2:-- Ueberwachungszeit KF1 hochfahren --, 3: VW_COMMENT
      ;ENDFOLD
      ;FOLD t8 ( EIN ) = -50[1/10Sek] ;%{SE}%MKUKATPVW %CVW_SPS %VTASG %P 2:t8 ( EIN ) = -50[1/10Sek], 3: TASG
         VW(#SET_TIME,TRUE,8,0,-50)
      ;ENDFOLD
      ;FOLD Schritt 121 = A4039 ;%{SE}%MKUKATPVW %CVW_SPS %VST_CON %P 2:Schritt 121 = A4039, 3: ST_CON
         IF $OUT[4039] THEN
            PREVSTEP = $APP_INT[5]
            $APP_INT[5] = 121
         ENDIF
      ;ENDFOLD
   ;ENDFOLD
   ;FOLD SCHRITT 121 -- ROB STP1 SZ1 -- ;%{P}%MKUKATPVW,%CSTEP,%VST_NR,%P 1:SCHRITT, 2:121, 3: ROB STP1 SZ1
      ;FOLD ;%{H}
         Case 121
      ;ENDFOLD
      ;FOLD -- Umdreh. KF setzen -- ;%{SE}%MKUKATPVW %CVW_COM %VCOMMENT %P 2:-- Umdreh. KF setzen --, 3: VW_COMMENT
      ;ENDFOLD
      ;FOLD i1 ( EIN ) = 0 ;%{SE}%MKUKATPVW %CVW_SPS %VARIASG %P 2:i1 ( EIN ) = 0, 3: ARIASG
         VW(#COUNTER,TRUE,1,0)
      ;ENDFOLD
      ;FOLD -- Ueberwachungszeit KF1 -- ;%{SE}%MKUKATPVW %CVW_COM %VCOMMENT %P 2:-- Ueberwachungszeit KF1 --, 3: VW_COMMENT
      ;ENDFOLD
      ;FOLD t7 ( EIN ) = -120[1/10Sek] ;%{SE}%MKUKATPVW %CVW_SPS %VTASG %P 2:t7 ( EIN ) = -120[1/10Sek], 3: TASG
         VW(#SET_TIME,TRUE,7,0,-120)
      ;ENDFOLD
      ;FOLD -- KF1 einschalten -- ;%{SE}%MKUKATPVW %CVW_COM %VCOMMENT %P 2:-- KF1 einschalten --, 3: VW_COMMENT
      ;ENDFOLD
      ;FOLD i1 (EIN) = 0 ;%{SE}%MKUKATPVW %CVW_SPS %VARIASG %P 2:i1 (EIN) = 0, 3: ARIASG
         VW(#COUNTER,TRUE,1,0)
      ;ENDFOLD
      ;FOLD A864 = EIN ;%{SE}%MKUKATPVW %CVW_SPS %VBOASG %P 2:A864 = EIN, 3: BOASG
         $OUT[864] = TRUE
      ;ENDFOLD
      ;FOLD -- KF1 hochfahren -- ;%{SE}%MKUKATPVW %CVW_COM %VCOMMENT %P 2:-- KF1 hochfahren --, 3: VW_COMMENT
      ;ENDFOLD
      ;FOLD A863 = EIN ;%{SE}%MKUKATPVW %CVW_SPS %VBOASG %P 2:A863 = EIN, 3: BOASG
         $OUT[863] = TRUE
      ;ENDFOLD
      ;FOLD Schritt 122 = (!E863 + T8) & A4039 ;%{SE}%MKUKATPVW %CVW_SPS %VST_CON %P 2:Schritt 122 = (!E863 + T8) & A4039, 3: ST_CON
         IF (NOT $IN[863] OR $TIMER_FLAG[8]) AND $OUT[4039] THEN
            PREVSTEP = $APP_INT[5]
            $APP_INT[5] = 122
         ENDIF
      ;ENDFOLD
   ;ENDFOLD
   ;FOLD SCHRITT 122 -- ROB STP1 SZ1 -- ;%{P}%MKUKATPVW,%CSTEP,%VST_NR,%P 1:SCHRITT, 2:122, 3: ROB STP1 SZ1
      ;FOLD ;%{H}
         Case 122
      ;ENDFOLD
      ;FOLD -- Funktionstest KF Motor -- ;%{SE}%MKUKATPVW %CVW_COM %VCOMMENT %P 2:-- Funktionstest KF Motor --, 3: VW_COMMENT
      ;ENDFOLD
      ;FOLD F312 = EIN ;%{SE}%MKUKATPVW %CVW_SPS %VBOASG %P 2:F312 = EIN, 3: BOASG
         $FLAG[312] = TRUE
      ;ENDFOLD
      ;FOLD F313 = i1 > 2 ;%{SE}%MKUKATPVW %CVW_SPS %VBOCMP %P 2:F313 = i1 > 2, 3: BOCMP
         $FLAG[313] = $COUNT_I[1] > 2
      ;ENDFOLD
      ;FOLD -- RSK Fehlerausgabe KF1 hochfahren -- ;%{SE}%MKUKATPVW %CVW_COM %VCOMMENT %P 2:-- RSK Fehlerausgabe KF1 hochfahren --, 3: VW_COMMENT
      ;ENDFOLD
      ;FOLD F324 = E863 + T8 + F324 ;%{SE}%MKUKATPVW %CVW_SPS %VBOASG %P 2:F324 = E863 + T8 + F324, 3: BOASG
         $FLAG[324] = $IN[863] OR $TIMER_FLAG[8] OR $FLAG[324]
      ;ENDFOLD
      ;FOLD Schritt 123 = (F313 + T7 + T8) & A4039 ;%{SE}%MKUKATPVW %CVW_SPS %VST_CON %P 2:Schritt 123 = (F313 + T7 + T8) & A4039, 3: ST_CON
         IF ($FLAG[313] OR $TIMER_FLAG[7] OR $TIMER_FLAG[8]) AND $OUT[4039] THEN
            PREVSTEP = $APP_INT[5]
            $APP_INT[5] = 123
         ENDIF
      ;ENDFOLD
   ;ENDFOLD
   ;FOLD SCHRITT 123 -- ROB STP1 SZ1 -- ;%{P}%MKUKATPVW,%CSTEP,%VST_NR,%P 1:SCHRITT, 2:123, 3: ROB STP1 SZ1
      ;FOLD ;%{H}
         Case 123
      ;ENDFOLD
      ;FOLD F312 = AUS ;%{SE}%MKUKATPVW %CVW_SPS %VBOASG %P 2:F312 = AUS, 3: BOASG
         $FLAG[312] = FALSE
